LIN {X 0,Y 249.241,Z 277.058,A -85,B 0,C 180,E1 -19068.615,E2 -19068.615} C_VEL
LIN {X 0,Y 249.451,Z 277.034,A -85,B 0,C 180,E1 -19071.901,E2 -19071.901} C_VEL
LIN {X 0,Y 249.292,Z 277.04,A -85,B 0,C 180,E1 -19075.148,E2 -19075.148} C_VEL
LIN {X 0,Y 249.563,Z 277.018,A -85,B 0,C 180,E1 -19077.813,E2 -19077.813} C_VEL
LIN {X 0,Y 249.011,Z 277.095,A -85,B 0,C 180,E1 -19079.16,E2 -19079.16} C_VEL
LIN {X 0,Y 247.389,Z 277.302,A -85,B 0,C 180,E1 -19080.48,E2 -19080.48} C_VEL
LIN {X 0,Y 243.426,Z 277.789,A -85,B 0,C 180,E1 -19083.136,E2 -19083.136} C_VEL
LIN {X 0,Y 242.327,Z 277.917,A -85,B 0,C 180,E1 -19084.528,E2 -19084.528} C_VEL
LIN {X 0,Y 242.256,Z 277.921,A -85,B 0,C 180,E1 -19085,E2 -19085} C_VEL
LIN {X 0,Y 242.423,Z 277.913,A -85,B 0,C 180,E1 -19088.334,E2 -19088.334} C_VEL
LIN {X 0,Y 242.16,Z 277.946,A -85,B 0,C 180,E1 -19093.425,E2 -19093.425} C_VEL
LIN {X 0,Y 242.146,Z 277.937,A -85,B 0,C 180,E1 -19096.872,E2 -19096.872} C_VEL
LIN {X 0,Y 242.049,Z 277.953,A -85,B 0,C 180,E1 -19101.703,E2 -19101.703} C_VEL
LIN {X 0,Y 242.063,Z 277.952,A -85,B 0,C 180,E1 -19105.838,E2 -19105.838} C_VEL
LIN {X 0,Y 242.003,Z 277.929,A -85,B 0,C 180,E1 -19109.583,E2 -19109.583} C_VEL
LIN {X 0,Y 241.984,Z 277.969,A -85,B 0,C 180,E1 -19113.492,E2 -19113.492} C_VEL
LIN {X 0,Y 241.987,Z 277.941,A -85,B 0,C 180,E1 -19117.582,E2 -19117.582} C_VEL
LIN {X 0,Y 241.966,Z 278.133,A -85,B 0,C 180,E1 -19122.089,E2 -19122.089} C_VEL
LIN {X 0,Y 244.588,Z 286.288,A -85,B 0,C 180,E1 -19125.918,E2 -19125.918} C_VEL
LIN {X 0,Y 246.843,Z 293.756,A -85,B 0,C 180,E1 -19129.093,E2 -19129.093} C_VEL
LIN {X 0,Y 249.068,Z 301.648,A -85,B 0,C 180,E1 -19132.141,E2 -19132.141} C_VEL
LIN {X 0,Y 255.279,Z 314.084,A -85,B 0,C 180,E1 -19133.592,E2 -19133.592} C_VEL
LIN {X 0,Y 262.138,Z 329.274,A -85,B 0,C 180,E1 -19135.107,E2 -19135.107} C_VEL
LIN {X 0,Y 263.614,Z 333.202,A -85,B 0,C 180,E1 -19135.441,E2 -19135.441} C_VEL
LIN {X 0,Y 264.453,Z 341.441,A -85,B 0,C 180,E1 -19135.825,E2 -19135.825} C_VEL
LIN {X 0,Y 260.682,Z 430.839,A -85,B 0,C 180,E1 -19138.284,E2 -19138.284} C_VEL
LIN {X 0,Y 259.42,Z 445.087,A -85,B 0,C 180,E1 -19138.965,E2 -19138.965} C_VEL
LIN {X 0,Y 257.726,Z 458.762,A -85,B 0,C 180,E1 -19139.93,E2 -19139.93} C_VEL
LIN {X 0,Y 255.853,Z 470.591,A -85,B 0,C 180,E1 -19141.045,E2 -19141.045} C_VEL
LIN {X 0,Y 253.532,Z 483.66,A -85,B 0,C 180,E1 -19142.644,E2 -19142.644} C_VEL
LIN {X 0,Y 251.02,Z 495.578,A -85,B 0,C 180,E1 -19144.504,E2 -19144.504} C_VEL
LIN {X 0,Y 248.301,Z 506.631,A -85,B 0,C 180,E1 -19146.656,E2 -19146.656} C_VEL
LIN {X 0,Y 245.98,Z 516.527,A -85,B 0,C 180,E1 -19149.076,E2 -19149.076} C_VEL
LIN {X 0,Y 244.075,Z 524.668,A -85,B 0,C 180,E1 -19151.535,E2 -19151.535} C_VEL
LIN {X 0,Y 242.606,Z 531.385,A -85,B 0,C 180,E1 -19154.026,E2 -19154.026} C_VEL
LIN {X 0,Y 241.38,Z 536.896,A -85,B 0,C 180,E1 -19156.531,E2 -19156.531} C_VEL
LIN {X 0,Y 240.535,Z 541.36,A -85,B 0,C 180,E1 -19159.052,E2 -19159.052} C_VEL
LIN {X 0,Y 240.083,Z 544.873,A -85,B 0,C 180,E1 -19161.584,E2 -19161.584} C_VEL
LIN {X 0,Y 239.765,Z 548.121,A -85,B 0,C 180,E1 -19164.955,E2 -19164.955} C_VEL
LIN {X 0,Y 239.831,Z 549.889,A -85,B 0,C 180,E1 -19168.321,E2 -19168.321} C_VEL
LIN {X 0,Y 239.891,Z 550.231,A -85,B 0,C 180,E1 -19170,E2 -19170} C_VEL
LIN {X 0,Y 239.832,Z 550.21,A -85,B 0,C 180,E1 -19171.679,E2 -19171.679} C_VEL
LIN {X 0,Y 239.798,Z 549.093,A -85,B 0,C 180,E1 -19175.044,E2 -19175.044} C_VEL
LIN {X 0,Y 240.089,Z 546.53,A -85,B 0,C 180,E1 -19178.416,E2 -19178.416} C_VEL
LIN {X 0,Y 240.843,Z 542.397,A -85,B 0,C 180,E1 -19181.786,E2 -19181.786} C_VEL
LIN {X 0,Y 242.35,Z 536.619,A -85,B 0,C 180,E1 -19185.129,E2 -19185.129} C_VEL
LIN {X 0,Y 243.804,Z 531.335,A -85,B 0,C 180,E1 -19187.509,E2 -19187.509} C_VEL
LIN {X 0,Y 245.627,Z 524.336,A -85,B 0,C 180,E1 -19190.081,E2 -19190.081} C_VEL
LIN {X 0,Y 247.967,Z 516.181,A -85,B 0,C 180,E1 -19192.496,E2 -19192.496} C_VEL
LIN {X 0,Y 250.678,Z 506.282,A -85,B 0,C 180,E1 -19194.868,E2 -19194.868} C_VEL
LIN {X 0,Y 253.686,Z 495.218,A -85,B 0,C 180,E1 -19196.977,E2 -19196.977} C_VEL
LIN {X 0,Y 256.269,Z 483.685,A -85,B 0,C 180,E1 -19198.752,E2 -19198.752} C_VEL
LIN {X 0,Y 258.66,Z 471.958,A -85,B 0,C 180,E1 -19200.176,E2 -19200.176} C_VEL
LIN {X 0,Y 260.838,Z 459.44,A -85,B 0,C 180,E1 -19201.356,E2 -19201.356} C_VEL
LIN {X 0,Y 262.802,Z 445.333,A -85,B 0,C 180,E1 -19202.333,E2 -19202.333} C_VEL
LIN {X 0,Y 264.18,Z 431.307,A -85,B 0,C 180,E1 -19202.992,E2 -19202.992} C_VEL
LIN {X 0,Y 266.368,Z 384.252,A -85,B 0,C 180,E1 -19204.294,E2 -19204.294} C_VEL
LIN {X 0,Y 268.154,Z 341.465,A -85,B 0,C 180,E1 -19205.452,E2 -19205.452} C_VEL
LIN {X 0,Y 267.344,Z 337.375,A -85,B 0,C 180,E1 -19205.711,E2 -19205.711} C_VEL
LIN {X 0,Y 259.951,Z 321.227,A -85,B 0,C 180,E1 -19207.443,E2 -19207.443} C_VEL
LIN {X 0,Y 253.336,Z 308.74,A -85,B 0,C 180,E1 -19209.035,E2 -19209.035} C_VEL
LIN {X 0,Y 249.464,Z 301.565,A -85,B 0,C 180,E1 -19210.088,E2 -19210.088} C_VEL
LIN {X 0,Y 247.111,Z 293.383,A -85,B 0,C 180,E1 -19213.557,E2 -19213.557} C_VEL
LIN {X 0,Y 244.395,Z 285.114,A -85,B 0,C 180,E1 -19217.486,E2 -19217.486} C_VEL
LIN {X 0,Y 241.98,Z 278.041,A -85,B 0,C 180,E1 -19221.315,E2 -19221.315} C_VEL
LIN {X 0,Y 241.979,Z 277.937,A -85,B 0,C 180,E1 -19224.488,E2 -19224.488} C_VEL
LIN {X 0,Y 241.969,Z 277.942,A -85,B 0,C 180,E1 -19228.48,E2 -19228.48} C_VEL
LIN {X 0,Y 241.999,Z 277.945,A -85,B 0,C 180,E1 -19232.312,E2 -19232.312} C_VEL
LIN {X 0,Y 242.054,Z 277.949,A -85,B 0,C 180,E1 -19236.016,E2 -19236.016} C_VEL
LIN {X 0,Y 242.034,Z 277.949,A -85,B 0,C 180,E1 -19239.608,E2 -19239.608} C_VEL
LIN {X 0,Y 242.16,Z 277.933,A -85,B 0,C 180,E1 -19243.278,E2 -19243.278} C_VEL
LIN {X 0,Y 242.183,Z 277.928,A -85,B 0,C 180,E1 -19248.28,E2 -19248.28} C_VEL
LIN {X 0,Y 242.423,Z 277.902,A -85,B 0,C 180,E1 -19251.666,E2 -19251.666} C_VEL
LIN {X 0,Y 242.256,Z 277.934,A -85,B 0,C 180,E1 -19255.008,E2 -19255.008} C_VEL
LIN {X 0,Y 242.633,Z 277.875,A -85,B 0,C 180,E1 -19258.341,E2 -19258.341} C_VEL
LIN {X 0,Y 242.633,Z 277.873,A -85,B 0,C 180,E1 -19261.66,E2 -19261.66} C_VEL
LIN {X 0,Y 242.425,Z 277.898,A -85,B 0,C 180,E1 -19266.74,E2 -19266.74} C_VEL
LIN {X 0,Y 242.312,Z 277.923,A -85,B 0,C 180,E1 -19270.022,E2 -19270.022} C_VEL
LIN {X 0,Y 242.162,Z 277.935,A -85,B 0,C 180,E1 -19275.142,E2 -19275.142} C_VEL
LIN {X 0,Y 242.071,Z 277.953,A -85,B 0,C 180,E1 -19278.625,E2 -19278.625} C_VEL
LIN {X 0,Y 242.04,Z 277.961,A -85,B 0,C 180,E1 -19282.178,E2 -19282.178} C_VEL
LIN {X 0,Y 242.065,Z 277.959,A -85,B 0,C 180,E1 -19285.839,E2 -19285.839} C_VEL
LIN {X 0,Y 242.006,Z 277.929,A -85,B 0,C 180,E1 -19289.584,E2 -19289.584} C_VEL
LIN {X 0,Y 241.99,Z 277.948,A -85,B 0,C 180,E1 -19293.492,E2 -19293.492} C_VEL
LIN {X 0,Y 242.04,Z 278.135,A -85,B 0,C 180,E1 -19296.725,E2 -19296.725} C_VEL
LIN {X 0,Y 244.197,Z 284.736,A -85,B 0,C 180,E1 -19300.358,E2 -19300.358} C_VEL
LIN {X 0,Y 246.509,Z 292.185,A -85,B 0,C 180,E1 -19304.056,E2 -19304.056} C_VEL
LIN {X 0,Y 248.881,Z 300.613,A -85,B 0,C 180,E1 -19307.84,E2 -19307.84} C_VEL
LIN {X 0,Y 251.042,Z 309.201,A -85,B 0,C 180,E1 -19311.295,E2 -19311.295} C_VEL
LIN {X 0,Y 255.898,Z 318.813,A -85,B 0,C 180,E1 -19312.553,E2 -19312.553} C_VEL
LIN {X 0,Y 262.144,Z 332.18,A -85,B 0,C 180,E1 -19314.035,E2 -19314.035} C_VEL
LIN {X 0,Y 265.974,Z 354.542,A -85,B 0,C 180,E1 -19315.331,E2 -19315.331} C_VEL
LIN {X 0,Y 267.064,Z 362.449,A -85,B 0,C 180,E1 -19315.736,E2 -19315.736} C_VEL
LIN {X 0,Y 264.429,Z 427.598,A -85,B 0,C 180,E1 -19317.384,E2 -19317.384} C_VEL
LIN {X 0,Y 263.126,Z 441.134,A -85,B 0,C 180,E1 -19317.994,E2 -19317.994} C_VEL
LIN {X 0,Y 261.559,Z 453.539,A -85,B 0,C 180,E1 -19318.853,E2 -19318.853} C_VEL
LIN {X 0,Y 259.621,Z 465.602,A -85,B 0,C 180,E1 -19319.993,E2 -19319.993} C_VEL
LIN {X 0,Y 257.248,Z 477.352,A -85,B 0,C 180,E1 -19321.439,E2 -19321.439} C_VEL
LIN {X 0,Y 254.58,Z 488.124,A -85,B 0,C 180,E1 -19323.125,E2 -19323.125} C_VEL
LIN {X 0,Y 252.112,Z 496.99,A -85,B 0,C 180,E1 -19324.842,E2 -19324.842} C_VEL
LIN {X 0,Y 249.235,Z 506.656,A -85,B 0,C 180,E1 -19327.187,E2 -19327.187} C_VEL
LIN {X 0,Y 246.739,Z 514.484,A -85,B 0,C 180,E1 -19329.579,E2 -19329.579} C_VEL
LIN {X 0,Y 244.494,Z 521.732,A -85,B 0,C 180,E1 -19332.433,E2 -19332.433} C_VEL
LIN {X 0,Y 242.871,Z 526.644,A -85,B 0,C 180,E1 -19334.904,E2 -19334.904} C_VEL
LIN {X 0,Y 241.633,Z 530.504,A -85,B 0,C 180,E1 -19337.4,E2 -19337.4} C_VEL
LIN {X 0,Y 240.832,Z 533.375,A -85,B 0,C 180,E1 -19339.916,E2 -19339.916} C_VEL
LIN {X 0,Y 240.401,Z 534.808,A -85,B 0,C 180,E1 -19341.595,E2 -19341.595} C_VEL
LIN {X 0,Y 239.927,Z 536.499,A -85,B 0,C 180,E1 -19344.959,E2 -19344.959} C_VEL
LIN {X 0,Y 239.893,Z 536.763,A -85,B 0,C 180,E1 -19348.321,E2 -19348.321} C_VEL
LIN {X 0,Y 240.021,Z 535.601,A -85,B 0,C 180,E1 -19351.678,E2 -19351.678} C_VEL
LIN {X 0,Y 240.545,Z 532.914,A -85,B 0,C 180,E1 -19355.028,E2 -19355.028} C_VEL
LIN {X 0,Y 241.466,Z 528.685,A -85,B 0,C 180,E1 -19358.368,E2 -19358.368} C_VEL
LIN {X 0,Y 242.501,Z 524.336,A -85,B 0,C 180,E1 -19360.858,E2 -19360.858} C_VEL
LIN {X 0,Y 244.235,Z 517.869,A -85,B 0,C 180,E1 -19363.733,E2 -19363.733} C_VEL
LIN {X 0,Y 246.174,Z 510.872,A -85,B 0,C 180,E1 -19366.161,E2 -19366.161} C_VEL
LIN {X 0,Y 248.461,Z 502.247,A -85,B 0,C 180,E1 -19368.555,E2 -19368.555} C_VEL
LIN {X 0,Y 250.585,Z 493.496,A -85,B 0,C 180,E1 -19370.522,E2 -19370.522} C_VEL
LIN {X 0,Y 253.083,Z 482.799,A -85,B 0,C 180,E1 -19372.447,E2 -19372.447} C_VEL
LIN {X 0,Y 255.272,Z 472.208,A -85,B 0,C 180,E1 -19373.959,E2 -19373.959} C_VEL
LIN {X 0,Y 257.329,Z 460.555,A -85,B 0,C 180,E1 -19375.26,E2 -19375.26} C_VEL
LIN {X 0,Y 259.046,Z 447.27,A -85,B 0,C 180,E1 -19376.38,E2 -19376.38} C_VEL
LIN {X 0,Y 260.309,Z 434.324,A -85,B 0,C 180,E1 -19377.14,E2 -19377.14} C_VEL
LIN {X 0,Y 261.113,Z 420.968,A -85,B 0,C 180,E1 -19377.622,E2 -19377.622} C_VEL
LIN {X 0,Y 263.267,Z 359.223,A -85,B 0,C 180,E1 -19379.182,E2 -19379.182} C_VEL
LIN {X 0,Y 258.935,Z 330.912,A -85,B 0,C 180,E1 -19380.645,E2 -19380.645} C_VEL
LIN {X 0,Y 257.727,Z 325.251,A -85,B 0,C 180,E1 -19380.995,E2 -19380.995} C_VEL
LIN {X 0,Y 251.935,Z 312.605,A -85,B 0,C 180,E1 -19382.282,E2 -19382.282} C_VEL
LIN {X 0,Y 250.406,Z 309.097,A -85,B 0,C 180,E1 -19382.745,E2 -19382.745} C_VEL
LIN {X 0,Y 248.171,Z 299.259,A -85,B 0,C 180,E1 -19386.491,E2 -19386.491} C_VEL
LIN {X 0,Y 246.195,Z 291.901,A -85,B 0,C 180,E1 -19389.577,E2 -19389.577} C_VEL
LIN {X 0,Y 243.774,Z 283.733,A -85,B 0,C 180,E1 -19393.283,E2 -19393.283} C_VEL
LIN {X 0,Y 241.929,Z 278.066,A -85,B 0,C 180,E1 -19396.14,E2 -19396.14} C_VEL
LIN {X 0,Y 241.972,Z 277.94,A -85,B 0,C 180,E1 -19400.283,E2 -19400.283} C_VEL
LIN {X 0,Y 242.036,Z 277.938,A -85,B 0,C 180,E1 -19404.497,E2 -19404.497} C_VEL
LIN {X 0,Y 241.974,Z 277.952,A -85,B 0,C 180,E1 -19408.479,E2 -19408.479} C_VEL
LIN {X 0,Y 242.005,Z 277.955,A -85,B 0,C 180,E1 -19412.312,E2 -19412.312} C_VEL
LIN {X 0,Y 242.055,Z 277.946,A -85,B 0,C 180,E1 -19416.015,E2 -19416.015} C_VEL
LIN {X 0,Y 242.034,Z 277.95,A -85,B 0,C 180,E1 -19419.607,E2 -19419.607} C_VEL
LIN {X 0,Y 242.161,Z 277.943,A -85,B 0,C 180,E1 -19423.277,E2 -19423.277} C_VEL
LIN {X 0,Y 242.177,Z 277.941,A -85,B 0,C 180,E1 -19428.279,E2 -19428.279} C_VEL
LIN {X 0,Y 242.397,Z 277.911,A -85,B 0,C 180,E1 -19431.664,E2 -19431.664} C_VEL
LIN {X 0,Y 242.252,Z 277.917,A -85,B 0,C 180,E1 -19435.006,E2 -19435.006} C_VEL
LIN {X 0,Y 242.632,Z 277.887,A -85,B 0,C 180,E1 -19438.34,E2 -19438.34} C_VEL
LIN {X 0,Y 242.632,Z 277.874,A -85,B 0,C 180,E1 -19441.659,E2 -19441.659} C_VEL
LIN {X 0,Y 242.256,Z 277.921,A -85,B 0,C 180,E1 -19445,E2 -19445} C_VEL
LIN {X 0,Y 241.632,Z 277.997,A -85,B 0,C 180,E1 -19446.39,E2 -19446.39} C_VEL
LIN {X 0,Y 238.772,Z 278.367,A -85,B 0,C 180,E1 -19448.656,E2 -19448.656} C_VEL
LIN {X 0,Y 236.291,Z 278.67,A -85,B 0,C 180,E1 -19450.502,E2 -19450.502} C_VEL
LIN {X 0,Y 235.197,Z 278.801,A -85,B 0,C 180,E1 -19451.935,E2 -19451.935} C_VEL
LIN {X 0,Y 235.093,Z 278.814,A -85,B 0,C 180,E1 -19452.422,E2 -19452.422} C_VEL
LIN {X 0,Y 235.092,Z 278.816,A -85,B 0,C 180,E1 -19456.94,E2 -19456.94} C_VEL
LIN {X 0,Y 234.989,Z 278.835,A -85,B 0,C 180,E1 -19462.01,E2 -19462.01} C_VEL
LIN {X 0,Y 234.964,Z 278.843,A -85,B 0,C 180,E1 -19466.657,E2 -19466.657} C_VEL
LIN {X 0,Y 234.918,Z 278.807,A -85,B 0,C 180,E1 -19470.569,E2 -19470.569} C_VEL
LIN {X 0,Y 234.938,Z 278.837,A -85,B 0,C 180,E1 -19474.636,E2 -19474.636} C_VEL
LIN {X 0,Y 234.938,Z 278.836,A -85,B 0,C 180,E1 -19478.945,E2 -19478.945} C_VEL
LIN {X 0,Y 234.927,Z 279,A -85,B 0,C 180,E1 -19480.591,E2 -19480.591} C_VEL
LIN {X 0,Y 237.675,Z 287.447,A -85,B 0,C 180,E1 -19484.793,E2 -19484.793} C_VEL
LIN {X 0,Y 240.055,Z 295.257,A -85,B 0,C 180,E1 -19488.291,E2 -19488.291} C_VEL
LIN {X 0,Y 241.831,Z 301.626,A -85,B 0,C 180,E1 -19490.881,E2 -19490.881} C_VEL
LIN {X 0,Y 247.567,Z 312.725,A -85,B 0,C 180,E1 -19492.326,E2 -19492.326} C_VEL
LIN {X 0,Y 254.203,Z 326.888,A -85,B 0,C 180,E1 -19493.87,E2 -19493.87} C_VEL
LIN {X 0,Y 257.787,Z 335.652,A -85,B 0,C 180,E1 -19494.701,E2 -19494.701} C_VEL
LIN {X 0,Y 258.422,Z 342.678,A -85,B 0,C 180,E1 -19495.029,E2 -19495.029} C_VEL
LIN {X 0,Y 254.549,Z 430.59,A -85,B 0,C 180,E1 -19497.485,E2 -19497.485} C_VEL
LIN {X 0,Y 253.26,Z 444.905,A -85,B 0,C 180,E1 -19498.181,E2 -19498.181} C_VEL
LIN {X 0,Y 251.586,Z 458.043,A -85,B 0,C 180,E1 -19499.117,E2 -19499.117} C_VEL
LIN {X 0,Y 249.633,Z 470.006,A -85,B 0,C 180,E1 -19500.252,E2 -19500.252} C_VEL
LIN {X 0,Y 247.517,Z 481.582,A -85,B 0,C 180,E1 -19501.668,E2 -19501.668} C_VEL
LIN {X 0,Y 245.128,Z 492.852,A -85,B 0,C 180,E1 -19503.386,E2 -19503.386} C_VEL
LIN {X 0,Y 242.729,Z 502.481,A -85,B 0,C 180,E1 -19505.176,E2 -19505.176} C_VEL
LIN {X 0,Y 240.071,Z 513.133,A -85,B 0,C 180,E1 -19507.631,E2 -19507.631} C_VEL
LIN {X 0,Y 237.898,Z 521.847,A -85,B 0,C 180,E1 -19510.14,E2 -19510.14} C_VEL
LIN {X 0,Y 236.051,Z 530.078,A -85,B 0,C 180,E1 -19513.125,E2 -19513.125} C_VEL
LIN {X 0,Y 234.448,Z 536.636,A -85,B 0,C 180,E1 -19516.125,E2 -19516.125} C_VEL
LIN {X 0,Y 233.513,Z 541.115,A -85,B 0,C 180,E1 -19518.719,E2 -19518.719} C_VEL
LIN {X 0,Y 233.032,Z 544.637,A -85,B 0,C 180,E1 -19521.327,E2 -19521.327} C_VEL
LIN {X 0,Y 232.686,Z 547.903,A -85,B 0,C 180,E1 -19524.801,E2 -19524.801} C_VEL
LIN {X 0,Y 232.742,Z 549.683,A -85,B 0,C 180,E1 -19528.27,E2 -19528.27} C_VEL
LIN {X 0,Y 232.801,Z 550.03,A -85,B 0,C 180,E1 -19530,E2 -19530} C_VEL
LIN {X 0,Y 232.743,Z 550.014,A -85,B 0,C 180,E1 -19531.73,E2 -19531.73} C_VEL
LIN {X 0,Y 232.727,Z 548.907,A -85,B 0,C 180,E1 -19535.198,E2 -19535.198} C_VEL
LIN {X 0,Y 233.04,Z 546.354,A -85,B 0,C 180,E1 -19538.673,E2 -19538.673} C_VEL
LIN {X 0,Y 233.603,Z 543.401,A -85,B 0,C 180,E1 -19541.277,E2 -19541.277} C_VEL
LIN {X 0,Y 234.994,Z 538.1,A -85,B 0,C 180,E1 -19544.727,E2 -19544.727} C_VEL
LIN {X 0,Y 236.798,Z 531.843,A -85,B 0,C 180,E1 -19547.758,E2 -19547.758} C_VEL
LIN {X 0,Y 238.911,Z 524.193,A -85,B 0,C 180,E1 -19550.671,E2 -19550.671} C_VEL
LIN {X 0,Y 241.367,Z 516.044,A -85,B 0,C 180,E1 -19553.146,E2 -19553.146} C_VEL
LIN {X 0,Y 244.241,Z 506.152,A -85,B 0,C 180,E1 -19555.57,E2 -19555.57} C_VEL
LIN {X 0,Y 247.364,Z 495.091,A -85,B 0,C 180,E1 -19557.725,E2 -19557.725} C_VEL
LIN {X 0,Y 249.938,Z 484.008,A -85,B 0,C 180,E1 -19559.477,E2 -19559.477} C_VEL
LIN {X 0,Y 252.55,Z 471.826,A -85,B 0,C 180,E1 -19560.985,E2 -19560.985} C_VEL
LIN {X 0,Y 254.787,Z 459.295,A -85,B 0,C 180,E1 -19562.188,E2 -19562.188} C_VEL
LIN {X 0,Y 256.833,Z 445.162,A -85,B 0,C 180,E1 -19563.18,E2 -19563.18} C_VEL
LIN {X 0,Y 258.231,Z 431.077,A -85,B 0,C 180,E1 -19563.853,E2 -19563.853} C_VEL
LIN {X 0,Y 260.282,Z 389.795,A -85,B 0,C 180,E1 -19565.009,E2 -19565.009} C_VEL
LIN {X 0,Y 262.345,Z 342.506,A -85,B 0,C 180,E1 -19566.312,E2 -19566.312} C_VEL
LIN {X 0,Y 261.526,Z 339.663,A -85,B 0,C 180,E1 -19566.54,E2 -19566.54} C_VEL
LIN {X 0,Y 254.828,Z 324.845,A -85,B 0,C 180,E1 -19568.186,E2 -19568.186} C_VEL
LIN {X 0,Y 248.582,Z 312.995,A -85,B 0,C 180,E1 -19569.755,E2 -19569.755} C_VEL
LIN {X 0,Y 242.373,Z 301.792,A -85,B 0,C 180,E1 -19571.473,E2 -19571.473} C_VEL
LIN {X 0,Y 239.793,Z 293.359,A -85,B 0,C 180,E1 -19575.3,E2 -19575.3} C_VEL
LIN {X 0,Y 237.206,Z 285.476,A -85,B 0,C 180,E1 -19579.321,E2 -19579.321} C_VEL
LIN {X 0,Y 234.941,Z 278.936,A -85,B 0,C 180,E1 -19583.12,E2 -19583.12} C_VEL
LIN {X 0,Y 234.952,Z 278.836,A -85,B 0,C 180,E1 -19587.424,E2 -19587.424} C_VEL
LIN {X 0,Y 234.933,Z 278.811,A -85,B 0,C 180,E1 -19591.404,E2 -19591.404} C_VEL
LIN {X 0,Y 234.983,Z 278.829,A -85,B 0,C 180,E1 -19595.247,E2 -19595.247} C_VEL
LIN {X 0,Y 235.008,Z 278.826,A -85,B 0,C 180,E1 -19598.97,E2 -19598.97} C_VEL
LIN {X 0,Y 235.093,Z 278.814,A -85,B 0,C 180,E1 -19603.06,E2 -19603.06} C_VEL
LIN {X 0,Y 235.115,Z 278.808,A -85,B 0,C 180,E1 -19607.923,E2 -19607.923} C_VEL
LIN {X 0,Y 235.372,Z 278.783,A -85,B 0,C 180,E1 -19611.414,E2 -19611.414} C_VEL
LIN {X 0,Y 235.399,Z 278.772,A -85,B 0,C 180,E1 -19613.142,E2 -19613.142} C_VEL
LIN {X 0,Y 235.592,Z 278.751,A -85,B 0,C 180,E1 -19618.291,E2 -19618.291} C_VEL
LIN {X 0,Y 235.593,Z 278.749,A -85,B 0,C 180,E1 -19621.71,E2 -19621.71} C_VEL
LIN {X 0,Y 235.401,Z 278.773,A -85,B 0,C 180,E1 -19626.859,E2 -19626.859} C_VEL
LIN {X 0,Y 235.235,Z 278.8,A -85,B 0,C 180,E1 -19630.327,E2 -19630.327} C_VEL
LIN {X 0,Y 235.11,Z 278.811,A -85,B 0,C 180,E1 -19635.607,E2 -19635.607} C_VEL
LIN {X 0,Y 235.007,Z 278.827,A -85,B 0,C 180,E1 -19639.206,E2 -19639.206} C_VEL
LIN {X 0,Y 234.974,Z 278.835,A -85,B 0,C 180,E1 -19642.882,E2 -19642.882} C_VEL
LIN {X 0,Y 234.966,Z 278.829,A -85,B 0,C 180,E1 -19646.659,E2 -19646.659} C_VEL
LIN {X 0,Y 234.922,Z 278.819,A -85,B 0,C 180,E1 -19650.57,E2 -19650.57} C_VEL
LIN {X 0,Y 234.994,Z 278.983,A -85,B 0,C 180,E1 -19654.883,E2 -19654.883} C_VEL
LIN {X 0,Y 236.993,Z 285.114,A -85,B 0,C 180,E1 -19658.518,E2 -19658.518} C_VEL
LIN {X 0,Y 239.386,Z 292.518,A -85,B 0,C 180,E1 -19662.474,E2 -19662.474} C_VEL
LIN {X 0,Y 241.579,Z 300.156,A -85,B 0,C 180,E1 -19666.12,E2 -19666.12} C_VEL
LIN {X 0,Y 243.828,Z 308.833,A -85,B 0,C 180,E1 -19669.854,E2 -19669.854} C_VEL
LIN {X 0,Y 246.07,Z 313.241,A -85,B 0,C 180,E1 -19670.55,E2 -19670.55} C_VEL
LIN {X 0,Y 251.385,Z 323.656,A -85,B 0,C 180,E1 -19671.923,E2 -19671.923} C_VEL
LIN {X 0,Y 256.825,Z 335.628,A -85,B 0,C 180,E1 -19673.274,E2 -19673.274} C_VEL
LIN {X 0,Y 260.897,Z 360.658,A -85,B 0,C 180,E1 -19674.742,E2 -19674.742} C_VEL
LIN {X 0,Y 261.153,Z 363.958,A -85,B 0,C 180,E1 -19674.887,E2 -19674.887} C_VEL
LIN {X 0,Y 258.462,Z 427.939,A -85,B 0,C 180,E1 -19676.543,E2 -19676.543} C_VEL
LIN {X 0,Y 257.142,Z 441.238,A -85,B 0,C 180,E1 -19677.157,E2 -19677.157} C_VEL
LIN {X 0,Y 255.51,Z 453.635,A -85,B 0,C 180,E1 -19678.03,E2 -19678.03} C_VEL
LIN {X 0,Y 253.384,Z 466.279,A -85,B 0,C 180,E1 -19679.252,E2 -19679.252} C_VEL
LIN {X 0,Y 251.049,Z 477.45,A -85,B 0,C 180,E1 -19680.666,E2 -19680.666} C_VEL
LIN {X 0,Y 248.242,Z 488.229,A -85,B 0,C 180,E1 -19682.381,E2 -19682.381} C_VEL
LIN {X 0,Y 245.166,Z 498.866,A -85,B 0,C 180,E1 -19684.533,E2 -19684.533} C_VEL
LIN {X 0,Y 242.225,Z 508.225,A -85,B 0,C 180,E1 -19686.94,E2 -19686.94} C_VEL
LIN {X 0,Y 239.672,Z 515.759,A -85,B 0,C 180,E1 -19689.398,E2 -19689.398} C_VEL
LIN {X 0,Y 237.682,Z 521.875,A -85,B 0,C 180,E1 -19691.912,E2 -19691.912} C_VEL
LIN {X 0,Y 236.015,Z 526.796,A -85,B 0,C 180,E1 -19694.455,E2 -19694.455} C_VEL
LIN {X 0,Y 234.684,Z 530.665,A -85,B 0,C 180,E1 -19697.021,E2 -19697.021} C_VEL
LIN {X 0,Y 233.806,Z 533.545,A -85,B 0,C 180,E1 -19699.61,E2 -19699.61} C_VEL
LIN {X 0,Y 233.361,Z 534.986,A -85,B 0,C 180,E1 -19701.339,E2 -19701.339} C_VEL
LIN {X 0,Y 232.849,Z 536.689,A -85,B 0,C 180,E1 -19704.805,E2 -19704.805} C_VEL
LIN {X 0,Y 232.806,Z 536.964,A -85,B 0,C 180,E1 -19708.27,E2 -19708.27} C_VEL
LIN {X 0,Y 232.935,Z 535.819,A -85,B 0,C 180,E1 -19711.729,E2 -19711.729} C_VEL
LIN {X 0,Y 233.488,Z 533.147,A -85,B 0,C 180,E1 -19715.181,E2 -19715.181} C_VEL
LIN {X 0,Y 234.458,Z 528.932,A -85,B 0,C 180,E1 -19718.62,E2 -19718.62} C_VEL
LIN {X 0,Y 235.529,Z 524.601,A -85,B 0,C 180,E1 -19721.183,E2 -19721.183} C_VEL
LIN {X 0,Y 237.345,Z 518.163,A -85,B 0,C 180,E1 -19724.14,E2 -19724.14} C_VEL
LIN {X 0,Y 239.371,Z 511.195,A -85,B 0,C 180,E1 -19726.634,E2 -19726.634} C_VEL
LIN {X 0,Y 241.749,Z 502.602,A -85,B 0,C 180,E1 -19729.09,E2 -19729.09} C_VEL
LIN {X 0,Y 243.985,Z 493.89,A -85,B 0,C 180,E1 -19731.104,E2 -19731.104} C_VEL
LIN {X 0,Y 246.573,Z 483.245,A -85,B 0,C 180,E1 -19733.073,E2 -19733.073} C_VEL
LIN {X 0,Y 248.835,Z 472.726,A -85,B 0,C 180,E1 -19734.619,E2 -19734.619} C_VEL
LIN {X 0,Y 250.955,Z 461.225,A -85,B 0,C 180,E1 -19735.949,E2 -19735.949} C_VEL
LIN {X 0,Y 252.669,Z 448.796,A -85,B 0,C 180,E1 -19737.044,E2 -19737.044} C_VEL
LIN {X 0,Y 254.016,Z 436.001,A -85,B 0,C 180,E1 -19737.842,E2 -19737.842} C_VEL
LIN {X 0,Y 254.918,Z 422.901,A -85,B 0,C 180,E1 -19738.357,E2 -19738.357} C_VEL
LIN {X 0,Y 257.196,Z 359.986,A -85,B 0,C 180,E1 -19739.993,E2 -19739.993} C_VEL
LIN {X 0,Y 253.075,Z 332.654,A -85,B 0,C 180,E1 -19741.455,E2 -19741.455} C_VEL
LIN {X 0,Y 252.068,Z 327.951,A -85,B 0,C 180,E1 -19741.759,E2 -19741.759} C_VEL
LIN {X 0,Y 246.262,Z 315.466,A -85,B 0,C 180,E1 -19743.103,E2 -19743.103} C_VEL
LIN {X 0,Y 243.307,Z 309.18,A -85,B 0,C 180,E1 -19743.885,E2 -19743.885} C_VEL
LIN {X 0,Y 241.436,Z 301.083,A -85,B 0,C 180,E1 -19747.055,E2 -19747.055} C_VEL
LIN {X 0,Y 239.476,Z 293.679,A -85,B 0,C 180,E1 -19750.266,E2 -19750.266} C_VEL
LIN {X 0,Y 236.754,Z 284.661,A -85,B 0,C 180,E1 -19754.565,E2 -19754.565} C_VEL
LIN {X 0,Y 234.904,Z 278.908,A -85,B 0,C 180,E1 -19757.675,E2 -19757.675} C_VEL
LIN {X 0,Y 234.955,Z 278.817,A -85,B 0,C 180,E1 -19761.085,E2 -19761.085} C_VEL
LIN {X 0,Y 234.96,Z 278.808,A -85,B 0,C 180,E1 -19765.366,E2 -19765.366} C_VEL
LIN {X 0,Y 234.967,Z 278.842,A -85,B 0,C 180,E1 -19770.157,E2 -19770.157} C_VEL
LIN {X 0,Y 234.992,Z 278.839,A -85,B 0,C 180,E1 -19773.793,E2 -19773.793} C_VEL
LIN {X 0,Y 235.009,Z 278.831,A -85,B 0,C 180,E1 -19778.969,E2 -19778.969} C_VEL
LIN {X 0,Y 235.094,Z 278.825,A -85,B 0,C 180,E1 -19783.059,E2 -19783.059} C_VEL
LIN {X 0,Y 235.11,Z 278.824,A -85,B 0,C 180,E1 -19787.921,E2 -19787.921} C_VEL
LIN {X 0,Y 235.328,Z 278.787,A -85,B 0,C 180,E1 -19791.412,E2 -19791.412} C_VEL
LIN {X 0,Y 235.389,Z 278.788,A -85,B 0,C 180,E1 -19793.14,E2 -19793.14} C_VEL
LIN {X 0,Y 235.591,Z 278.765,A -85,B 0,C 180,E1 -19798.29,E2 -19798.29} C_VEL
LIN {X 0,Y 235.592,Z 278.751,A -85,B 0,C 180,E1 -19801.709,E2 -19801.709} C_VEL
LIN {X 0,Y 235.4,Z 278.774,A -85,B 0,C 180,E1 -19806.858,E2 -19806.858} C_VEL
LIN {X 0,Y 235.234,Z 278.794,A -85,B 0,C 180,E1 -19810.326,E2 -19810.326} C_VEL
LIN {X 0,Y 235.093,Z 278.814,A -85,B 0,C 180,E1 -19812.422,E2 -19812.422} C_VEL
LIN {X 0,Y 234.387,Z 278.915,A -85,B 0,C 180,E1 -19813.852,E2 -19813.852} C_VEL
LIN {X 0,Y 231.517,Z 279.268,A -85,B 0,C 180,E1 -19816.186,E2 -19816.186} C_VEL
LIN {X 0,Y 229.087,Z 279.574,A -85,B 0,C 180,E1 -19818.089,E2 -19818.089} C_VEL
LIN {X 0,Y 228.025,Z 279.698,A -85,B 0,C 180,E1 -19819.565,E2 -19819.565} C_VEL
LIN {X 0,Y 227.927,Z 279.707,A -85,B 0,C 180,E1 -19820.066,E2 -19820.066} C_VEL
LIN {X 0,Y 227.91,Z 279.715,A -85,B 0,C 180,E1 -19823.633,E2 -19823.633} C_VEL
LIN {X 0,Y 227.876,Z 279.719,A -85,B 0,C 180,E1 -19827.556,E2 -19827.556} C_VEL
LIN {X 0,Y 227.864,Z 279.692,A -85,B 0,C 180,E1 -19831.623,E2 -19831.623} C_VEL
LIN {X 0,Y 227.879,Z 279.698,A -85,B 0,C 180,E1 -19835.871,E2 -19835.871} C_VEL
LIN {X 0,Y 227.928,Z 279.96,A -85,B 0,C 180,E1 -19839.016,E2 -19839.016} C_VEL
LIN {X 0,Y 230.916,Z 289.1,A -85,B 0,C 180,E1 -19843.819,E2 -19843.819} C_VEL
LIN {X 0,Y 233.177,Z 296.389,A -85,B 0,C 180,E1 -19847.268,E2 -19847.268} C_VEL
LIN {X 0,Y 234.73,Z 301.974,A -85,B 0,C 180,E1 -19849.607,E2 -19849.607} C_VEL
LIN {X 0,Y 241.502,Z 314.663,A -85,B 0,C 180,E1 -19851.369,E2 -19851.369} C_VEL
LIN {X 0,Y 248.702,Z 329.96,A -85,B 0,C 180,E1 -19853.124,E2 -19853.124} C_VEL
LIN {X 0,Y 251.971,Z 337.774,A -85,B 0,C 180,E1 -19853.909,E2 -19853.909} C_VEL
LIN {X 0,Y 252.44,Z 343.76,A -85,B 0,C 180,E1 -19854.188,E2 -19854.188} C_VEL
LIN {X 0,Y 248.47,Z 430.334,A -85,B 0,C 180,E1 -19856.648,E2 -19856.648} C_VEL
LIN {X 0,Y 247.249,Z 443.966,A -85,B 0,C 180,E1 -19857.312,E2 -19857.312} C_VEL
LIN {X 0,Y 245.662,Z 456.191,A -85,B 0,C 180,E1 -19858.166,E2 -19858.166} C_VEL
LIN {X 0,Y 243.469,Z 469.423,A -85,B 0,C 180,E1 -19859.419,E2 -19859.419} C_VEL
LIN {X 0,Y 241.043,Z 482.136,A -85,B 0,C 180,E1 -19861.009,E2 -19861.009} C_VEL
LIN {X 0,Y 238.485,Z 493.609,A -85,B 0,C 180,E1 -19862.821,E2 -19862.821} C_VEL
LIN {X 0,Y 235.737,Z 504.074,A -85,B 0,C 180,E1 -19864.86,E2 -19864.86} C_VEL
LIN {X 0,Y 233.057,Z 514.358,A -85,B 0,C 180,E1 -19867.389,E2 -19867.389} C_VEL
LIN {X 0,Y 230.827,Z 522.808,A -85,B 0,C 180,E1 -19869.969,E2 -19869.969} C_VEL
LIN {X 0,Y 228.926,Z 530.828,A -85,B 0,C 180,E1 -19873.044,E2 -19873.044} C_VEL
LIN {X 0,Y 227.5,Z 536.375,A -85,B 0,C 180,E1 -19875.692,E2 -19875.692} C_VEL
LIN {X 0,Y 226.509,Z 540.87,A -85,B 0,C 180,E1 -19878.365,E2 -19878.365} C_VEL
LIN {X 0,Y 225.975,Z 544.4,A -85,B 0,C 180,E1 -19881.054,E2 -19881.054} C_VEL
LIN {X 0,Y 225.733,Z 546.241,A -85,B 0,C 180,E1 -19882.846,E2 -19882.846} C_VEL
LIN {X 0,Y 225.55,Z 548.76,A -85,B 0,C 180,E1 -19886.427,E2 -19886.427} C_VEL
LIN {X 0,Y 225.636,Z 549.476,A -85,B 0,C 180,E1 -19888.215,E2 -19888.215} C_VEL
LIN {X 0,Y 225.714,Z 549.829,A -85,B 0,C 180,E1 -19890,E2 -19890} C_VEL
LIN {X 0,Y 225.637,Z 549.817,A -85,B 0,C 180,E1 -19891.785,E2 -19891.785} C_VEL
LIN {X 0,Y 225.64,Z 548.72,A -85,B 0,C 180,E1 -19895.362,E2 -19895.362} C_VEL
LIN {X 0,Y 225.986,Z 546.178,A -85,B 0,C 180,E1 -19898.946,E2 -19898.946} C_VEL
LIN {X 0,Y 226.594,Z 543.232,A -85,B 0,C 180,E1 -19901.631,E2 -19901.631} C_VEL
LIN {X 0,Y 228.084,Z 537.941,A -85,B 0,C 180,E1 -19905.183,E2 -19905.183} C_VEL
LIN {X 0,Y 230.115,Z 531.066,A -85,B 0,C 180,E1 -19908.573,E2 -19908.573} C_VEL
LIN {X 0,Y 232.628,Z 522.802,A -85,B 0,C 180,E1 -19911.721,E2 -19911.721} C_VEL
LIN {X 0,Y 235.297,Z 514.405,A -85,B 0,C 180,E1 -19914.248,E2 -19914.248} C_VEL
LIN {X 0,Y 238.43,Z 504.207,A -85,B 0,C 180,E1 -19916.712,E2 -19916.712} C_VEL
LIN {X 0,Y 241.373,Z 493.828,A -85,B 0,C 180,E1 -19918.713,E2 -19918.713} C_VEL
LIN {X 0,Y 244.007,Z 482.89,A -85,B 0,C 180,E1 -19920.435,E2 -19920.435} C_VEL
LIN {X 0,Y 246.809,Z 469.926,A -85,B 0,C 180,E1 -19922.029,E2 -19922.029} C_VEL
LIN {X 0,Y 249.188,Z 456.901,A -85,B 0,C 180,E1 -19923.244,E2 -19923.244} C_VEL
LIN {X 0,Y 251.238,Z 442.717,A -85,B 0,C 180,E1 -19924.2,E2 -19924.2} C_VEL
LIN {X 0,Y 252.485,Z 429.653,A -85,B 0,C 180,E1 -19924.793,E2 -19924.793} C_VEL
LIN {X 0,Y 256.557,Z 345.746,A -85,B 0,C 180,E1 -19927.138,E2 -19927.138} C_VEL
LIN {X 0,Y 256.471,Z 343.541,A -85,B 0,C 180,E1 -19927.231,E2 -19927.231} C_VEL
LIN {X 0,Y 249.83,Z 328.641,A -85,B 0,C 180,E1 -19928.939,E2 -19928.939} C_VEL
LIN {X 0,Y 242.408,Z 314.491,A -85,B 0,C 180,E1 -19930.902,E2 -19930.902} C_VEL
LIN {X 0,Y 237.027,Z 305.289,A -85,B 0,C 180,E1 -19932.398,E2 -19932.398} C_VEL
LIN {X 0,Y 235.191,Z 301.931,A -85,B 0,C 180,E1 -19933.019,E2 -19933.019} C_VEL
LIN {X 0,Y 233.036,Z 294.954,A -85,B 0,C 180,E1 -19936.368,E2 -19936.368} C_VEL
LIN {X 0,Y 230.635,Z 287.822,A -85,B 0,C 180,E1 -19940.215,E2 -19940.215} C_VEL
LIN {X 0,Y 228.273,Z 281.258,A -85,B 0,C 180,E1 -19944.2,E2 -19944.2} C_VEL
LIN {X 0,Y 227.893,Z 279.794,A -85,B 0,C 180,E1 -19945.214,E2 -19945.214} C_VEL
LIN {X 0,Y 227.901,Z 279.68,A -85,B 0,C 180,E1 -19950.436,E2 -19950.436} C_VEL
LIN {X 0,Y 227.925,Z 279.714,A -85,B 0,C 180,E1 -19954.426,E2 -19954.426} C_VEL
LIN {X 0,Y 227.959,Z 279.709,A -85,B 0,C 180,E1 -19958.287,E2 -19958.287} C_VEL
LIN {X 0,Y 228.031,Z 279.695,A -85,B 0,C 180,E1 -19962.826,E2 -19962.826} C_VEL
LIN {X 0,Y 228.072,Z 279.687,A -85,B 0,C 180,E1 -19967.544,E2 -19967.544} C_VEL
LIN {X 0,Y 228.302,Z 279.667,A -85,B 0,C 180,E1 -19971.146,E2 -19971.146} C_VEL
LIN {X 0,Y 228.35,Z 279.649,A -85,B 0,C 180,E1 -19972.929,E2 -19972.929} C_VEL
LIN {X 0,Y 228.551,Z 279.628,A -85,B 0,C 180,E1 -19978.238,E2 -19978.238} C_VEL
LIN {X 0,Y 228.551,Z 279.626,A -85,B 0,C 180,E1 -19981.763,E2 -19981.763} C_VEL
LIN {X 0,Y 228.352,Z 279.65,A -85,B 0,C 180,E1 -19987.072,E2 -19987.072} C_VEL
LIN {X 0,Y 228.157,Z 279.678,A -85,B 0,C 180,E1 -19990.651,E2 -19990.651} C_VEL
LIN {X 0,Y 228.061,Z 279.699,A -85,B 0,C 180,E1 -19994.273,E2 -19994.273} C_VEL
LIN {X 0,Y 228.001,Z 279.71,A -85,B 0,C 180,E1 -19997.954,E2 -19997.954} C_VEL
LIN {X 0,Y 227.952,Z 279.715,A -85,B 0,C 180,E1 -20002.344,E2 -20002.344} C_VEL
LIN {X 0,Y 227.941,Z 279.703,A -85,B 0,C 180,E1 -20006.603,E2 -20006.603} C_VEL
LIN {X 0,Y 227.896,Z 279.69,A -85,B 0,C 180,E1 -20010.292,E2 -20010.292} C_VEL
LIN {X 0,Y 227.96,Z 279.941,A -85,B 0,C 180,E1 -20012.915,E2 -20012.915} C_VEL
LIN {X 0,Y 230.022,Z 285.881,A -85,B 0,C 180,E1 -20016.751,E2 -20016.751} C_VEL
LIN {X 0,Y 232.284,Z 293.112,A -85,B 0,C 180,E1 -20020.853,E2 -20020.853} C_VEL
LIN {X 0,Y 234.59,Z 300.745,A -85,B 0,C 180,E1 -20024.751,E2 -20024.751} C_VEL
LIN {X 0,Y 236.735,Z 308.899,A -85,B 0,C 180,E1 -20028.425,E2 -20028.425} C_VEL
LIN {X 0,Y 244.381,Z 323.185,A -85,B 0,C 180,E1 -20030.59,E2 -20030.59} C_VEL
LIN {X 0,Y 251.338,Z 338.057,A -85,B 0,C 180,E1 -20032.407,E2 -20032.407} C_VEL
LIN {X 0,Y 255.13,Z 361.799,A -85,B 0,C 180,E1 -20033.85,E2 -20033.85} C_VEL
LIN {X 0,Y 255.351,Z 365.68,A -85,B 0,C 180,E1 -20034.013,E2 -20034.013} C_VEL
LIN {X 0,Y 252.618,Z 427.25,A -85,B 0,C 180,E1 -20035.621,E2 -20035.621} C_VEL
LIN {X 0,Y 251.333,Z 440.574,A -85,B 0,C 180,E1 -20036.237,E2 -20036.237} C_VEL
LIN {X 0,Y 249.51,Z 453.731,A -85,B 0,C 180,E1 -20037.166,E2 -20037.166} C_VEL
LIN {X 0,Y 247.499,Z 465.329,A -85,B 0,C 180,E1 -20038.296,E2 -20038.296} C_VEL
LIN {X 0,Y 245.221,Z 476.168,A -85,B 0,C 180,E1 -20039.66,E2 -20039.66} C_VEL
LIN {X 0,Y 242.319,Z 487.27,A -85,B 0,C 180,E1 -20041.41,E2 -20041.41} C_VEL
LIN {X 0,Y 239.303,Z 497.214,A -85,B 0,C 180,E1 -20043.393,E2 -20043.393} C_VEL
LIN {X 0,Y 236.212,Z 506.895,A -85,B 0,C 180,E1 -20045.852,E2 -20045.852} C_VEL
LIN {X 0,Y 233.415,Z 514.742,A -85,B 0,C 180,E1 -20048.356,E2 -20048.356} C_VEL
LIN {X 0,Y 231.575,Z 520.106,A -85,B 0,C 180,E1 -20050.498,E2 -20050.498} C_VEL
LIN {X 0,Y 229.722,Z 525.412,A -85,B 0,C 180,E1 -20053.104,E2 -20053.104} C_VEL
LIN {X 0,Y 228.098,Z 529.623,A -85,B 0,C 180,E1 -20055.73,E2 -20055.73} C_VEL
LIN {X 0,Y 226.801,Z 533.714,A -85,B 0,C 180,E1 -20059.285,E2 -20059.285} C_VEL
LIN {X 0,Y 226.32,Z 535.163,A -85,B 0,C 180,E1 -20061.068,E2 -20061.068} C_VEL
LIN {X 0,Y 225.773,Z 536.879,A -85,B 0,C 180,E1 -20064.642,E2 -20064.642} C_VEL
LIN {X 0,Y 225.72,Z 537.166,A -85,B 0,C 180,E1 -20068.216,E2 -20068.216} C_VEL
LIN {X 0,Y 225.852,Z 536.037,A -85,B 0,C 180,E1 -20071.783,E2 -20071.783} C_VEL
LIN {X 0,Y 226.435,Z 533.38,A -85,B 0,C 180,E1 -20075.343,E2 -20075.343} C_VEL
LIN {X 0,Y 227.441,Z 529.18,A -85,B 0,C 180,E1 -20078.888,E2 -20078.888} C_VEL
LIN {X 0,Y 228.579,Z 524.866,A -85,B 0,C 180,E1 -20081.528,E2 -20081.528} C_VEL
LIN {X 0,Y 230.483,Z 518.454,A -85,B 0,C 180,E1 -20084.57,E2 -20084.57} C_VEL
LIN {X 0,Y 232.592,Z 511.518,A -85,B 0,C 180,E1 -20087.134,E2 -20087.134} C_VEL
LIN {X 0,Y 235.069,Z 502.956,A -85,B 0,C 180,E1 -20089.654,E2 -20089.654} C_VEL
LIN {X 0,Y 237.409,Z 494.284,A -85,B 0,C 180,E1 -20091.717,E2 -20091.717} C_VEL
LIN {X 0,Y 240.08,Z 483.692,A -85,B 0,C 180,E1 -20093.735,E2 -20093.735} C_VEL
LIN {X 0,Y 242.434,Z 473.243,A -85,B 0,C 180,E1 -20095.314,E2 -20095.314} C_VEL
LIN {X 0,Y 244.608,Z 461.86,A -85,B 0,C 180,E1 -20096.675,E2 -20096.675} C_VEL
LIN {X 0,Y 246.339,Z 450.231,A -85,B 0,C 180,E1 -20097.746,E2 -20097.746} C_VEL
LIN {X 0,Y 247.799,Z 437.363,A -85,B 0,C 180,E1 -20098.594,E2 -20098.594} C_VEL
LIN {X 0,Y 248.814,Z 423.411,A -85,B 0,C 180,E1 -20099.174,E2 -20099.174} C_VEL
LIN {X 0,Y 251.208,Z 360.984,A -85,B 0,C 180,E1 -20100.83,E2 -20100.83} C_VEL
LIN {X 0,Y 246.894,Z 331.846,A -85,B 0,C 180,E1 -20102.446,E2 -20102.446} C_VEL
LIN {X 0,Y 241.623,Z 320.228,A -85,B 0,C 180,E1 -20103.725,E2 -20103.725} C_VEL
LIN {X 0,Y 236.19,Z 309.016,A -85,B 0,C 180,E1 -20105.169,E2 -20105.169} C_VEL
LIN {X 0,Y 234.164,Z 300.475,A -85,B 0,C 180,E1 -20108.707,E2 -20108.707} C_VEL
LIN {X 0,Y 231.961,Z 292.755,A -85,B 0,C 180,E1 -20112.304,E2 -20112.304} C_VEL
LIN {X 0,Y 230.085,Z 286.718,A -85,B 0,C 180,E1 -20115.368,E2 -20115.368} C_VEL
LIN {X 0,Y 227.865,Z 279.784,A -85,B 0,C 180,E1 -20119.31,E2 -20119.31} C_VEL
LIN {X 0,Y 227.899,Z 279.703,A -85,B 0,C 180,E1 -20124.131,E2 -20124.131} C_VEL
LIN {X 0,Y 227.871,Z 279.704,A -85,B 0,C 180,E1 -20128.377,E2 -20128.377} C_VEL
LIN {X 0,Y 227.884,Z 279.715,A -85,B 0,C 180,E1 -20132.444,E2 -20132.444} C_VEL
LIN {X 0,Y 227.912,Z 279.708,A -85,B 0,C 180,E1 -20136.366,E2 -20136.366} C_VEL
LIN {X 0,Y 227.94,Z 279.703,A -85,B 0,C 180,E1 -20140.174,E2 -20140.174} C_VEL
LIN {X 0,Y 228.054,Z 279.693,A -85,B 0,C 180,E1 -20143.897,E2 -20143.897} C_VEL
LIN {X 0,Y 228.068,Z 279.701,A -85,B 0,C 180,E1 -20147.542,E2 -20147.542} C_VEL
LIN {X 0,Y 228.264,Z 279.664,A -85,B 0,C 180,E1 -20151.144,E2 -20151.144} C_VEL
LIN {X 0,Y 228.336,Z 279.668,A -85,B 0,C 180,E1 -20152.927,E2 -20152.927} C_VEL
LIN {X 0,Y 228.55,Z 279.642,A -85,B 0,C 180,E1 -20158.237,E2 -20158.237} C_VEL
LIN {X 0,Y 228.551,Z 279.628,A -85,B 0,C 180,E1 -20161.762,E2 -20161.762} C_VEL
LIN {X 0,Y 228.351,Z 279.654,A -85,B 0,C 180,E1 -20167.071,E2 -20167.071} C_VEL
LIN {X 0,Y 228.155,Z 279.674,A -85,B 0,C 180,E1 -20170.65,E2 -20170.65} C_VEL
LIN {X 0,Y 228.059,Z 279.699,A -85,B 0,C 180,E1 -20174.272,E2 -20174.272} C_VEL
LIN {X 0,Y 227.999,Z 279.709,A -85,B 0,C 180,E1 -20177.953,E2 -20177.953} C_VEL
LIN {X 0,Y 227.927,Z 279.707,A -85,B 0,C 180,E1 -20180.066,E2 -20180.066} C_VEL
LIN {X 0,Y 227.23,Z 279.799,A -85,B 0,C 180,E1 -20181.54,E2 -20181.54} C_VEL
LIN {X 0,Y 224.378,Z 280.16,A -85,B 0,C 180,E1 -20183.946,E2 -20183.946} C_VEL
LIN {X 0,Y 221.965,Z 280.463,A -85,B 0,C 180,E1 -20185.908,E2 -20185.908} C_VEL
LIN {X 0,Y 220.919,Z 280.586,A -85,B 0,C 180,E1 -20187.432,E2 -20187.432} C_VEL
LIN {X 0,Y 220.827,Z 280.584,A -85,B 0,C 180,E1 -20187.948,E2 -20187.948} C_VEL
LIN {X 0,Y 220.835,Z 280.561,A -85,B 0,C 180,E1 -20190.768,E2 -20190.768} C_VEL
LIN {X 0,Y 220.8,Z 280.59,A -85,B 0,C 180,E1 -20194.955,E2 -20194.955} C_VEL
LIN {X 0,Y 220.848,Z 280.826,A -85,B 0,C 180,E1 -20197.202,E2 -20197.202} C_VEL
LIN {X 0,Y 223.283,Z 288.098,A -85,B 0,C 180,E1 -20201.375,E2 -20201.375} C_VEL
LIN {X 0,Y 225.953,Z 296.519,A -85,B 0,C 180,E1 -20205.674,E2 -20205.674} C_VEL
LIN {X 0,Y 227.608,Z 302.185,A -85,B 0,C 180,E1 -20208.197,E2 -20208.197} C_VEL
LIN {X 0,Y 234.644,Z 315.005,A -85,B 0,C 180,E1 -20210.141,E2 -20210.141} C_VEL
LIN {X 0,Y 242.198,Z 330.697,A -85,B 0,C 180,E1 -20212.081,E2 -20212.081} C_VEL
LIN {X 0,Y 246.27,Z 340.399,A -85,B 0,C 180,E1 -20213.109,E2 -20213.109} C_VEL
LIN {X 0,Y 246.511,Z 344.831,A -85,B 0,C 180,E1 -20213.307,E2 -20213.307} C_VEL
LIN {X 0,Y 242.448,Z 430.067,A -85,B 0,C 180,E1 -20215.769,E2 -20215.769} C_VEL
LIN {X 0,Y 241.198,Z 443.783,A -85,B 0,C 180,E1 -20216.448,E2 -20216.448} C_VEL
LIN {X 0,Y 239.459,Z 456.602,A -85,B 0,C 180,E1 -20217.365,E2 -20217.365} C_VEL
LIN {X 0,Y 237.355,Z 468.838,A -85,B 0,C 180,E1 -20218.543,E2 -20218.543} C_VEL
LIN {X 0,Y 234.785,Z 481.803,A -85,B 0,C 180,E1 -20220.187,E2 -20220.187} C_VEL
LIN {X 0,Y 232.133,Z 493.178,A -85,B 0,C 180,E1 -20222.014,E2 -20222.014} C_VEL
LIN {X 0,Y 229.304,Z 503.695,A -85,B 0,C 180,E1 -20224.104,E2 -20224.104} C_VEL
LIN {X 0,Y 226.91,Z 512.446,A -85,B 0,C 180,E1 -20226.257,E2 -20226.257} C_VEL
LIN {X 0,Y 224.459,Z 521.226,A -85,B 0,C 180,E1 -20228.896,E2 -20228.896} C_VEL
LIN {X 0,Y 222.568,Z 528.456,A -85,B 0,C 180,E1 -20231.593,E2 -20231.593} C_VEL
LIN {X 0,Y 221.033,Z 534.395,A -85,B 0,C 180,E1 -20234.32,E2 -20234.32} C_VEL
LIN {X 0,Y 219.774,Z 539.221,A -85,B 0,C 180,E1 -20237.065,E2 -20237.065} C_VEL
LIN {X 0,Y 218.937,Z 544.163,A -85,B 0,C 180,E1 -20240.764,E2 -20240.764} C_VEL
LIN {X 0,Y 218.499,Z 547.466,A -85,B 0,C 180,E1 -20244.463,E2 -20244.463} C_VEL
LIN {X 0,Y 218.532,Z 549.268,A -85,B 0,C 180,E1 -20248.157,E2 -20248.157} C_VEL
LIN {X 0,Y 218.629,Z 549.628,A -85,B 0,C 180,E1 -20250,E2 -20250} C_VEL
LIN {X 0,Y 218.497,Z 549.256,A -85,B 0,C 180,E1 -20253.688,E2 -20253.688} C_VEL
LIN {X 0,Y 218.561,Z 548.534,A -85,B 0,C 180,E1 -20255.536,E2 -20255.536} C_VEL
LIN {X 0,Y 218.949,Z 546.001,A -85,B 0,C 180,E1 -20259.236,E2 -20259.236} C_VEL
LIN {X 0,Y 219.875,Z 541.902,A -85,B 0,C 180,E1 -20262.929,E2 -20262.929} C_VEL
LIN {X 0,Y 221.189,Z 537.782,A -85,B 0,C 180,E1 -20265.669,E2 -20265.669} C_VEL
LIN {X 0,Y 222.864,Z 532.607,A -85,B 0,C 180,E1 -20268.382,E2 -20268.382} C_VEL
LIN {X 0,Y 225.189,Z 525.154,A -85,B 0,C 180,E1 -20271.513,E2 -20271.513} C_VEL
LIN {X 0,Y 227.814,Z 517.275,A -85,B 0,C 180,E1 -20274.127,E2 -20274.127} C_VEL
LIN {X 0,Y 230.89,Z 507.691,A -85,B 0,C 180,E1 -20276.677,E2 -20276.677} C_VEL
LIN {X 0,Y 233.887,Z 498.069,A -85,B 0,C 180,E1 -20278.736,E2 -20278.736} C_VEL
LIN {X 0,Y 236.901,Z 486.628,A -85,B 0,C 180,E1 -20280.73,E2 -20280.73} C_VEL
LIN {X 0,Y 239.739,Z 474.848,A -85,B 0,C 180,E1 -20282.344,E2 -20282.344} C_VEL
LIN {X 0,Y 242.493,Z 461.223,A -85,B 0,C 180,E1 -20283.786,E2 -20283.786} C_VEL
LIN {X 0,Y 244.669,Z 447.856,A -85,B 0,C 180,E1 -20284.812,E2 -20284.812} C_VEL
LIN {X 0,Y 246.321,Z 433.999,A -85,B 0,C 180,E1 -20285.544,E2 -20285.544} C_VEL
LIN {X 0,Y 247.471,Z 416.592,A -85,B 0,C 180,E1 -20286.106,E2 -20286.106} C_VEL
LIN {X 0,Y 250.808,Z 345.883,A -85,B 0,C 180,E1 -20288.12,E2 -20288.12} C_VEL
LIN {X 0,Y 244.15,Z 330.905,A -85,B 0,C 180,E1 -20289.92,E2 -20289.92} C_VEL
LIN {X 0,Y 236.701,Z 316.893,A -85,B 0,C 180,E1 -20291.993,E2 -20291.993} C_VEL
LIN {X 0,Y 230.735,Z 306.623,A -85,B 0,C 180,E1 -20293.762,E2 -20293.762} C_VEL
LIN {X 0,Y 228.108,Z 302.208,A -85,B 0,C 180,E1 -20294.642,E2 -20294.642} C_VEL
LIN {X 0,Y 225.365,Z 293.699,A -85,B 0,C 180,E1 -20299.09,E2 -20299.09} C_VEL
LIN {X 0,Y 223.006,Z 286.805,A -85,B 0,C 180,E1 -20303.218,E2 -20303.218} C_VEL
LIN {X 0,Y 221.815,Z 283.416,A -85,B 0,C 180,E1 -20305.464,E2 -20305.464} C_VEL
LIN {X 0,Y 220.813,Z 280.681,A -85,B 0,C 180,E1 -20307.515,E2 -20307.515} C_VEL
LIN {X 0,Y 220.824,Z 280.567,A -85,B 0,C 180,E1 -20311.485,E2 -20311.485} C_VEL
LIN {X 0,Y 220.864,Z 280.587,A -85,B 0,C 180,E1 -20315.565,E2 -20315.565} C_VEL
LIN {X 0,Y 220.889,Z 280.582,A -85,B 0,C 180,E1 -20319.514,E2 -20319.514} C_VEL
LIN {X 0,Y 221.013,Z 280.566,A -85,B 0,C 180,E1 -20323.371,E2 -20323.371} C_VEL
LIN {X 0,Y 221.104,Z 280.555,A -85,B 0,C 180,E1 -20329.006,E2 -20329.006} C_VEL
LIN {X 0,Y 221.285,Z 280.529,A -85,B 0,C 180,E1 -20332.702,E2 -20332.702} C_VEL
LIN {X 0,Y 221.509,Z 280.504,A -85,B 0,C 180,E1 -20338.182,E2 -20338.182} C_VEL
LIN {X 0,Y 221.51,Z 280.502,A -85,B 0,C 180,E1 -20341.819,E2 -20341.819} C_VEL
LIN {X 0,Y 221.287,Z 280.53,A -85,B 0,C 180,E1 -20347.299,E2 -20347.299} C_VEL
LIN {X 0,Y 221.104,Z 280.554,A -85,B 0,C 180,E1 -20350.995,E2 -20350.995} C_VEL
LIN {X 0,Y 221.014,Z 280.568,A -85,B 0,C 180,E1 -20356.631,E2 -20356.631} C_VEL
LIN {X 0,Y 220.898,Z 280.583,A -85,B 0,C 180,E1 -20360.486,E2 -20360.486} C_VEL
LIN {X 0,Y 220.87,Z 280.589,A -85,B 0,C 180,E1 -20364.435,E2 -20364.435} C_VEL
LIN {X 0,Y 220.826,Z 280.564,A -85,B 0,C 180,E1 -20368.516,E2 -20368.516} C_VEL
LIN {X 0,Y 220.868,Z 280.803,A -85,B 0,C 180,E1 -20370.606,E2 -20370.606} C_VEL
LIN {X 0,Y 222.905,Z 286.347,A -85,B 0,C 180,E1 -20374.579,E2 -20374.579} C_VEL
LIN {X 0,Y 224.593,Z 291.623,A -85,B 0,C 180,E1 -20377.869,E2 -20377.869} C_VEL
LIN {X 0,Y 226.831,Z 298.878,A -85,B 0,C 180,E1 -20381.962,E2 -20381.962} C_VEL
LIN {X 0,Y 228.814,Z 306,A -85,B 0,C 180,E1 -20385.572,E2 -20385.572} C_VEL
LIN {X 0,Y 229.681,Z 308.972,A -85,B 0,C 180,E1 -20386.853,E2 -20386.853} C_VEL
LIN {X 0,Y 237.584,Z 323.326,A -85,B 0,C 180,E1 -20389.218,E2 -20389.218} C_VEL
LIN {X 0,Y 243.151,Z 334.696,A -85,B 0,C 180,E1 -20390.77,E2 -20390.77} C_VEL
LIN {X 0,Y 246.123,Z 341.578,A -85,B 0,C 180,E1 -20391.581,E2 -20391.581} C_VEL
LIN {X 0,Y 249.675,Z 364.685,A -85,B 0,C 180,E1 -20393.019,E2 -20393.019} C_VEL
LIN {X 0,Y 246.798,Z 427.62,A -85,B 0,C 180,E1 -20394.703,E2 -20394.703} C_VEL
LIN {X 0,Y 245.371,Z 441.451,A -85,B 0,C 180,E1 -20395.364,E2 -20395.364} C_VEL
LIN {X 0,Y 243.397,Z 454.962,A -85,B 0,C 180,E1 -20396.356,E2 -20396.356} C_VEL
LIN {X 0,Y 241.33,Z 466.232,A -85,B 0,C 180,E1 -20397.501,E2 -20397.501} C_VEL
LIN {X 0,Y 238.784,Z 477.647,A -85,B 0,C 180,E1 -20398.998,E2 -20398.998} C_VEL
LIN {X 0,Y 235.752,Z 488.437,A -85,B 0,C 180,E1 -20400.781,E2 -20400.781} C_VEL
LIN {X 0,Y 232.403,Z 499.089,A -85,B 0,C 180,E1 -20403.025,E2 -20403.025} C_VEL
LIN {X 0,Y 229.204,Z 508.47,A -85,B 0,C 180,E1 -20405.547,E2 -20405.547} C_VEL
LIN {X 0,Y 226.396,Z 516.025,A -85,B 0,C 180,E1 -20408.13,E2 -20408.13} C_VEL
LIN {X 0,Y 224.149,Z 522.161,A -85,B 0,C 180,E1 -20410.779,E2 -20410.779} C_VEL
LIN {X 0,Y 222.307,Z 527.102,A -85,B 0,C 180,E1 -20413.47,E2 -20413.47} C_VEL
LIN {X 0,Y 220.786,Z 530.989,A -85,B 0,C 180,E1 -20416.188,E2 -20416.188} C_VEL
LIN {X 0,Y 219.813,Z 533.883,A -85,B 0,C 180,E1 -20418.94,E2 -20418.94} C_VEL
LIN {X 0,Y 219.298,Z 535.34,A -85,B 0,C 180,E1 -20420.779,E2 -20420.779} C_VEL
LIN {X 0,Y 218.699,Z 537.07,A -85,B 0,C 180,E1 -20424.468,E2 -20424.468} C_VEL
LIN {X 0,Y 218.635,Z 537.367,A -85,B 0,C 180,E1 -20428.158,E2 -20428.158} C_VEL
LIN {X 0,Y 218.771,Z 536.253,A -85,B 0,C 180,E1 -20431.841,E2 -20431.841} C_VEL
LIN {X 0,Y 219.365,Z 533.613,A -85,B 0,C 180,E1 -20435.515,E2 -20435.515} C_VEL
LIN {X 0,Y 220.44,Z 529.428,A -85,B 0,C 180,E1 -20439.172,E2 -20439.172} C_VEL
LIN {X 0,Y 221.651,Z 525.13,A -85,B 0,C 180,E1 -20441.893,E2 -20441.893} C_VEL
LIN {X 0,Y 223.644,Z 518.741,A -85,B 0,C 180,E1 -20445.026,E2 -20445.026} C_VEL
LIN {X 0,Y 225.832,Z 511.837,A -85,B 0,C 180,E1 -20447.663,E2 -20447.663} C_VEL
LIN {X 0,Y 228.418,Z 503.309,A -85,B 0,C 180,E1 -20450.251,E2 -20450.251} C_VEL
LIN {X 0,Y 230.86,Z 494.676,A -85,B 0,C 180,E1 -20452.366,E2 -20452.366} C_VEL
LIN {X 0,Y 233.626,Z 484.137,A -85,B 0,C 180,E1 -20454.433,E2 -20454.433} C_VEL
LIN {X 0,Y 236.059,Z 473.757,A -85,B 0,C 180,E1 -20456.048,E2 -20456.048} C_VEL
LIN {X 0,Y 238.31,Z 462.473,A -85,B 0,C 180,E1 -20457.438,E2 -20457.438} C_VEL
LIN {X 0,Y 240.281,Z 449.716,A -85,B 0,C 180,E1 -20458.637,E2 -20458.637} C_VEL
LIN {X 0,Y 241.8,Z 436.8,A -85,B 0,C 180,E1 -20459.486,E2 -20459.486} C_VEL
LIN {X 0,Y 242.785,Z 423.859,A -85,B 0,C 180,E1 -20460.031,E2 -20460.031} C_VEL
LIN {X 0,Y 245.277,Z 361.947,A -85,B 0,C 180,E1 -20461.709,E2 -20461.709} C_VEL
LIN {X 0,Y 241.237,Z 334.404,A -85,B 0,C 180,E1 -20463.298,E2 -20463.298} C_VEL
LIN {X 0,Y 235.042,Z 320.823,A -85,B 0,C 180,E1 -20464.883,E2 -20464.883} C_VEL
LIN {X 0,Y 229.074,Z 308.862,A -85,B 0,C 180,E1 -20466.554,E2 -20466.554} C_VEL
LIN {X 0,Y 227.415,Z 302.27,A -85,B 0,C 180,E1 -20469.411,E2 -20469.411} C_VEL
LIN {X 0,Y 225.107,Z 294.103,A -85,B 0,C 180,E1 -20473.38,E2 -20473.38} C_VEL
LIN {X 0,Y 222.564,Z 286.123,A -85,B 0,C 180,E1 -20477.725,E2 -20477.725} C_VEL
LIN {X 0,Y 220.823,Z 280.676,A -85,B 0,C 180,E1 -20481.055,E2 -20481.055} C_VEL
LIN {X 0,Y 220.819,Z 280.564,A -85,B 0,C 180,E1 -20485.841,E2 -20485.841} C_VEL
LIN {X 0,Y 220.867,Z 280.596,A -85,B 0,C 180,E1 -20489.394,E2 -20489.394} C_VEL
LIN {X 0,Y 220.893,Z 280.596,A -85,B 0,C 180,E1 -20493.548,E2 -20493.548} C_VEL
LIN {X 0,Y 220.876,Z 280.595,A -85,B 0,C 180,E1 -20497.552,E2 -20497.552} C_VEL
LIN {X 0,Y 220.982,Z 280.584,A -85,B 0,C 180,E1 -20502.57,E2 -20502.57} C_VEL
LIN {X 0,Y 221.007,Z 280.58,A -85,B 0,C 180,E1 -20507.138,E2 -20507.138} C_VEL
LIN {X 0,Y 221.201,Z 280.541,A -85,B 0,C 180,E1 -20510.859,E2 -20510.859} C_VEL
LIN {X 0,Y 221.268,Z 280.55,A -85,B 0,C 180,E1 -20512.7,E2 -20512.7} C_VEL
LIN {X 0,Y 221.508,Z 280.52,A -85,B 0,C 180,E1 -20518.181,E2 -20518.181} C_VEL
LIN {X 0,Y 221.509,Z 280.506,A -85,B 0,C 180,E1 -20521.818,E2 -20521.818} C_VEL
LIN {X 0,Y 221.286,Z 280.535,A -85,B 0,C 180,E1 -20527.298,E2 -20527.298} C_VEL
LIN {X 0,Y 221.103,Z 280.551,A -85,B 0,C 180,E1 -20530.994,E2 -20530.994} C_VEL
LIN {X 0,Y 221.012,Z 280.567,A -85,B 0,C 180,E1 -20536.63,E2 -20536.63} C_VEL
LIN {X 0,Y 220.889,Z 280.582,A -85,B 0,C 180,E1 -20540.486,E2 -20540.486} C_VEL
LIN {X 0,Y 220.863,Z 280.587,A -85,B 0,C 180,E1 -20544.435,E2 -20544.435} C_VEL
LIN {X 0,Y 220.827,Z 280.584,A -85,B 0,C 180,E1 -20547.948,E2 -20547.948} C_VEL
LIN {X 0,Y 220.127,Z 280.657,A -85,B 0,C 180,E1 -20548.959,E2 -20548.959} C_VEL
LIN {X 0,Y 217.257,Z 281.007,A -85,B 0,C 180,E1 -20550.546,E2 -20550.546} C_VEL
LIN {X 0,Y 214.385,Z 281.376,A -85,B 0,C 180,E1 -20552.173,E2 -20552.173} C_VEL
LIN {X 0,Y 213.724,Z 281.472,A -85,B 0,C 180,E1 -20553.23,E2 -20553.23} C_VEL
LIN {X 0,Y 213.789,Z 281.699,A -85,B 0,C 180,E1 -20555.194,E2 -20555.194} C_VEL
LIN {X 0,Y 216.085,Z 288.328,A -85,B 0,C 180,E1 -20559.36,E2 -20559.36} C_VEL
LIN {X 0,Y 218.639,Z 296.22,A -85,B 0,C 180,E1 -20563.717,E2 -20563.717} C_VEL
LIN {X 0,Y 220.469,Z 302.309,A -85,B 0,C 180,E1 -20566.652,E2 -20566.652} C_VEL
LIN {X 0,Y 227.946,Z 315.623,A -85,B 0,C 180,E1 -20568.86,E2 -20568.86} C_VEL
LIN {X 0,Y 234.506,Z 328.783,A -85,B 0,C 180,E1 -20570.646,E2 -20570.646} C_VEL
LIN {X 0,Y 240.58,Z 342.836,A -85,B 0,C 180,E1 -20572.257,E2 -20572.257} C_VEL
LIN {X 0,Y 240.505,Z 348.913,A -85,B 0,C 180,E1 -20572.471,E2 -20572.471} C_VEL
LIN {X 0,Y 236.488,Z 429.789,A -85,B 0,C 180,E1 -20574.846,E2 -20574.846} C_VEL
LIN {X 0,Y 235.193,Z 443.598,A -85,B 0,C 180,E1 -20575.537,E2 -20575.537} C_VEL
LIN {X 0,Y 233.446,Z 455.876,A -85,B 0,C 180,E1 -20576.415,E2 -20576.415} C_VEL
LIN {X 0,Y 231.282,Z 468.252,A -85,B 0,C 180,E1 -20577.618,E2 -20577.618} C_VEL
LIN {X 0,Y 228.807,Z 480.291,A -85,B 0,C 180,E1 -20579.144,E2 -20579.144} C_VEL
LIN {X 0,Y 225.826,Z 492.747,A -85,B 0,C 180,E1 -20581.16,E2 -20581.16} C_VEL
LIN {X 0,Y 222.912,Z 503.315,A -85,B 0,C 180,E1 -20583.303,E2 -20583.303} C_VEL
LIN {X 0,Y 220.381,Z 512.102,A -85,B 0,C 180,E1 -20585.508,E2 -20585.508} C_VEL
LIN {X 0,Y 217.784,Z 520.911,A -85,B 0,C 180,E1 -20588.216,E2 -20588.216} C_VEL
LIN {X 0,Y 215.523,Z 529.237,A -85,B 0,C 180,E1 -20591.462,E2 -20591.462} C_VEL
LIN {X 0,Y 213.671,Z 535.852,A -85,B 0,C 180,E1 -20594.744,E2 -20594.744} C_VEL
LIN {X 0,Y 212.504,Z 540.379,A -85,B 0,C 180,E1 -20597.587,E2 -20597.587} C_VEL
LIN {X 0,Y 211.876,Z 543.924,A -85,B 0,C 180,E1 -20600.454,E2 -20600.454} C_VEL
LIN {X 0,Y 211.595,Z 545.788,A -85,B 0,C 180,E1 -20602.365,E2 -20602.365} C_VEL
LIN {X 0,Y 211.349,Z 548.335,A -85,B 0,C 180,E1 -20606.187,E2 -20606.187} C_VEL
LIN {X 0,Y 211.43,Z 549.061,A -85,B 0,C 180,E1 -20608.095,E2 -20608.095} C_VEL
LIN {X 0,Y 211.545,Z 549.427,A -85,B 0,C 180,E1 -20610,E2 -20610} C_VEL
LIN {X 0,Y 211.415,Z 549.065,A -85,B 0,C 180,E1 -20613.812,E2 -20613.812} C_VEL
LIN {X 0,Y 211.609,Z 547.268,A -85,B 0,C 180,E1 -20617.634,E2 -20617.634} C_VEL
LIN {X 0,Y 212.331,Z 543.987,A -85,B 0,C 180,E1 -20621.455,E2 -20621.455} C_VEL
LIN {X 0,Y 213.807,Z 539.081,A -85,B 0,C 180,E1 -20625.246,E2 -20625.246} C_VEL
LIN {X 0,Y 215.443,Z 534.298,A -85,B 0,C 180,E1 -20628.053,E2 -20628.053} C_VEL
LIN {X 0,Y 217.749,Z 527.286,A -85,B 0,C 180,E1 -20631.29,E2 -20631.29} C_VEL
LIN {X 0,Y 220.815,Z 518.528,A -85,B 0,C 180,E1 -20634.441,E2 -20634.441} C_VEL
LIN {X 0,Y 223.954,Z 509.302,A -85,B 0,C 180,E1 -20637.066,E2 -20637.066} C_VEL
LIN {X 0,Y 227.356,Z 499.019,A -85,B 0,C 180,E1 -20639.388,E2 -20639.388} C_VEL
LIN {X 0,Y 230.55,Z 487.54,A -85,B 0,C 180,E1 -20641.468,E2 -20641.468} C_VEL
LIN {X 0,Y 233.76,Z 474.723,A -85,B 0,C 180,E1 -20643.276,E2 -20643.276} C_VEL
LIN {X 0,Y 236.631,Z 461.09,A -85,B 0,C 180,E1 -20644.741,E2 -20644.741} C_VEL
LIN {X 0,Y 238.877,Z 447.694,A -85,B 0,C 180,E1 -20645.784,E2 -20645.784} C_VEL
LIN {X 0,Y 240.563,Z 433.783,A -85,B 0,C 180,E1 -20646.53,E2 -20646.53} C_VEL
LIN {X 0,Y 241.878,Z 414.556,A -85,B 0,C 180,E1 -20647.143,E2 -20647.143} C_VEL
LIN {X 0,Y 245.166,Z 348.069,A -85,B 0,C 180,E1 -20649.064,E2 -20649.064} C_VEL
LIN {X 0,Y 237.851,Z 331.923,A -85,B 0,C 180,E1 -20651.141,E2 -20651.141} C_VEL
LIN {X 0,Y 229.352,Z 316.078,A -85,B 0,C 180,E1 -20653.677,E2 -20653.677} C_VEL
LIN {X 0,Y 223.214,Z 306.272,A -85,B 0,C 180,E1 -20655.628,E2 -20655.628} C_VEL
LIN {X 0,Y 220.881,Z 302.279,A -85,B 0,C 180,E1 -20656.524,E2 -20656.524} C_VEL
LIN {X 0,Y 218.588,Z 295.194,A -85,B 0,C 180,E1 -20660.501,E2 -20660.501} C_VEL
LIN {X 0,Y 216.135,Z 287.944,A -85,B 0,C 180,E1 -20665.163,E2 -20665.163} C_VEL
LIN {X 0,Y 213.793,Z 281.61,A -85,B 0,C 180,E1 -20670.071,E2 -20670.071} C_VEL
LIN {X 0,Y 213.823,Z 281.455,A -85,B 0,C 180,E1 -20672.603,E2 -20672.603} C_VEL
LIN {X 0,Y 213.849,Z 281.468,A -85,B 0,C 180,E1 -20676.953,E2 -20676.953} C_VEL
LIN {X 0,Y 213.941,Z 281.45,A -85,B 0,C 180,E1 -20682.804,E2 -20682.804} C_VEL
LIN {X 0,Y 213.951,Z 281.452,A -85,B 0,C 180,E1 -20686.707,E2 -20686.707} C_VEL
LIN {X 0,Y 214.164,Z 281.433,A -85,B 0,C 180,E1 -20690.557,E2 -20690.557} C_VEL
LIN {X 0,Y 214.223,Z 281.409,A -85,B 0,C 180,E1 -20692.46,E2 -20692.46} C_VEL
LIN {X 0,Y 214.442,Z 281.383,A -85,B 0,C 180,E1 -20698.123,E2 -20698.123} C_VEL
LIN {X 0,Y 214.547,Z 281.386,A -85,B 0,C 180,E1 -20700.001,E2 -20700.001} C_VEL
LIN {X 0,Y 214.443,Z 281.382,A -85,B 0,C 180,E1 -20701.879,E2 -20701.879} C_VEL
LIN {X 0,Y 214.225,Z 281.41,A -85,B 0,C 180,E1 -20707.541,E2 -20707.541} C_VEL
LIN {X 0,Y 214.021,Z 281.435,A -85,B 0,C 180,E1 -20711.364,E2 -20711.364} C_VEL
LIN {X 0,Y 213.93,Z 281.449,A -85,B 0,C 180,E1 -20715.238,E2 -20715.238} C_VEL
LIN {X 0,Y 213.84,Z 281.463,A -85,B 0,C 180,E1 -20719.188,E2 -20719.188} C_VEL
LIN {X 0,Y 213.853,Z 281.463,A -85,B 0,C 180,E1 -20723.227,E2 -20723.227} C_VEL
LIN {X 0,Y 213.822,Z 281.618,A -85,B 0,C 180,E1 -20727.936,E2 -20727.936} C_VEL
LIN {X 0,Y 215.925,Z 287.34,A -85,B 0,C 180,E1 -20732.483,E2 -20732.483} C_VEL
LIN {X 0,Y 217.993,Z 293.433,A -85,B 0,C 180,E1 -20736.615,E2 -20736.615} C_VEL
LIN {X 0,Y 220.123,Z 300.628,A -85,B 0,C 180,E1 -20740.883,E2 -20740.883} C_VEL
LIN {X 0,Y 222.35,Z 308.405,A -85,B 0,C 180,E1 -20744.962,E2 -20744.962} C_VEL
LIN {X 0,Y 225.163,Z 313.308,A -85,B 0,C 180,E1 -20745.961,E2 -20745.961} C_VEL
LIN {X 0,Y 233.211,Z 327.977,A -85,B 0,C 180,E1 -20748.46,E2 -20748.46} C_VEL
LIN {X 0,Y 238.863,Z 339.812,A -85,B 0,C 180,E1 -20750.106,E2 -20750.106} C_VEL
LIN {X 0,Y 240.893,Z 344.61,A -85,B 0,C 180,E1 -20750.687,E2 -20750.687} C_VEL
LIN {X 0,Y 244.016,Z 366.093,A -85,B 0,C 180,E1 -20752.051,E2 -20752.051} C_VEL
LIN {X 0,Y 241.109,Z 427.133,A -85,B 0,C 180,E1 -20753.707,E2 -20753.707} C_VEL
LIN {X 0,Y 239.674,Z 440.788,A -85,B 0,C 180,E1 -20754.353,E2 -20754.353} C_VEL
LIN {X 0,Y 237.714,Z 453.924,A -85,B 0,C 180,E1 -20755.311,E2 -20755.311} C_VEL
LIN {X 0,Y 235.384,Z 466.327,A -85,B 0,C 180,E1 -20756.574,E2 -20756.574} C_VEL
LIN {X 0,Y 232.657,Z 478.033,A -85,B 0,C 180,E1 -20758.144,E2 -20758.144} C_VEL
LIN {X 0,Y 229.591,Z 488.541,A -85,B 0,C 180,E1 -20759.918,E2 -20759.918} C_VEL
LIN {X 0,Y 226.071,Z 499.202,A -85,B 0,C 180,E1 -20762.205,E2 -20762.205} C_VEL
LIN {X 0,Y 222.755,Z 508.592,A -85,B 0,C 180,E1 -20764.791,E2 -20764.791} C_VEL
LIN {X 0,Y 219.797,Z 516.158,A -85,B 0,C 180,E1 -20767.437,E2 -20767.437} C_VEL
LIN {X 0,Y 217.43,Z 522.304,A -85,B 0,C 180,E1 -20770.16,E2 -20770.16} C_VEL
LIN {X 0,Y 215.483,Z 527.255,A -85,B 0,C 180,E1 -20772.93,E2 -20772.93} C_VEL
LIN {X 0,Y 213.871,Z 531.149,A -85,B 0,C 180,E1 -20775.732,E2 -20775.732} C_VEL
LIN {X 0,Y 212.812,Z 534.052,A -85,B 0,C 180,E1 -20778.571,E2 -20778.571} C_VEL
LIN {X 0,Y 212.268,Z 535.517,A -85,B 0,C 180,E1 -20780.471,E2 -20780.471} C_VEL
LIN {X 0,Y 211.641,Z 537.26,A -85,B 0,C 180,E1 -20784.283,E2 -20784.283} C_VEL
LIN {X 0,Y 211.534,Z 537.569,A -85,B 0,C 180,E1 -20788.096,E2 -20788.096} C_VEL
LIN {X 0,Y 211.692,Z 536.468,A -85,B 0,C 180,E1 -20791.902,E2 -20791.902} C_VEL
LIN {X 0,Y 211.95,Z 535.348,A -85,B 0,C 180,E1 -20793.802,E2 -20793.802} C_VEL
LIN {X 0,Y 212.777,Z 531.962,A -85,B 0,C 180,E1 -20797.592,E2 -20797.592} C_VEL
LIN {X 0,Y 213.82,Z 528.36,A -85,B 0,C 180,E1 -20800.415,E2 -20800.415} C_VEL
LIN {X 0,Y 215.253,Z 523.737,A -85,B 0,C 180,E1 -20803.211,E2 -20803.211} C_VEL
LIN {X 0,Y 217.539,Z 516.863,A -85,B 0,C 180,E1 -20806.42,E2 -20806.42} C_VEL
LIN {X 0,Y 219.937,Z 509.497,A -85,B 0,C 180,E1 -20809.119,E2 -20809.119} C_VEL
LIN {X 0,Y 222.763,Z 500.441,A -85,B 0,C 180,E1 -20811.759,E2 -20811.759} C_VEL
LIN {X 0,Y 225.715,Z 490.101,A -85,B 0,C 180,E1 -20814.121,E2 -20814.121} C_VEL
LIN {X 0,Y 228.363,Z 479.693,A -85,B 0,C 180,E1 -20816.011,E2 -20816.011} C_VEL
LIN {X 0,Y 231.027,Z 468.211,A -85,B 0,C 180,E1 -20817.639,E2 -20817.639} C_VEL
LIN {X 0,Y 233.266,Z 456.432,A -85,B 0,C 180,E1 -20818.932,E2 -20818.932} C_VEL
LIN {X 0,Y 234.94,Z 443.939,A -85,B 0,C 180,E1 -20819.97,E2 -20819.97} C_VEL
LIN {X 0,Y 236.394,Z 430.402,A -85,B 0,C 180,E1 -20820.703,E2 -20820.703} C_VEL
LIN {X 0,Y 237.332,Z 412.874,A -85,B 0,C 180,E1 -20821.258,E2 -20821.258} C_VEL
LIN {X 0,Y 239.314,Z 362.022,A -85,B 0,C 180,E1 -20822.677,E2 -20822.677} C_VEL
LIN {X 0,Y 235.624,Z 336.96,A -85,B 0,C 180,E1 -20824.192,E2 -20824.192} C_VEL
LIN {X 0,Y 228.647,Z 321.704,A -85,B 0,C 180,E1 -20826.079,E2 -20826.079} C_VEL
LIN {X 0,Y 223.248,Z 311.542,A -85,B 0,C 180,E1 -20827.593,E2 -20827.593} C_VEL
LIN {X 0,Y 221.818,Z 308.438,A -85,B 0,C 180,E1 -20828.149,E2 -20828.149} C_VEL
LIN {X 0,Y 219.55,Z 299.87,A -85,B 0,C 180,E1 -20832.238,E2 -20832.238} C_VEL
LIN {X 0,Y 217.496,Z 293.038,A -85,B 0,C 180,E1 -20835.891,E2 -20835.891} C_VEL
LIN {X 0,Y 215.652,Z 287.176,A -85,B 0,C 180,E1 -20839.322,E2 -20839.322} C_VEL
LIN {X 0,Y 213.78,Z 281.562,A -85,B 0,C 180,E1 -20843.031,E2 -20843.031} C_VEL
LIN {X 0,Y 213.767,Z 281.441,A -85,B 0,C 180,E1 -20846.019,E2 -20846.019} C_VEL
LIN {X 0,Y 213.779,Z 281.476,A -85,B 0,C 180,E1 -20850.453,E2 -20850.453} C_VEL
LIN {X 0,Y 213.8,Z 281.47,A -85,B 0,C 180,E1 -20854.701,E2 -20854.701} C_VEL
LIN {X 0,Y 213.811,Z 281.472,A -85,B 0,C 180,E1 -20858.802,E2 -20858.802} C_VEL
LIN {X 0,Y 213.941,Z 281.461,A -85,B 0,C 180,E1 -20862.803,E2 -20862.803} C_VEL
LIN {X 0,Y 213.949,Z 281.454,A -85,B 0,C 180,E1 -20866.706,E2 -20866.706} C_VEL
LIN {X 0,Y 214.139,Z 281.419,A -85,B 0,C 180,E1 -20870.554,E2 -20870.554} C_VEL
LIN {X 0,Y 214.205,Z 281.428,A -85,B 0,C 180,E1 -20872.458,E2 -20872.458} C_VEL
LIN {X 0,Y 214.441,Z 281.4,A -85,B 0,C 180,E1 -20878.121,E2 -20878.121} C_VEL
LIN {X 0,Y 214.546,Z 281.369,A -85,B 0,C 180,E1 -20879.999,E2 -20879.999} C_VEL
LIN {X 0,Y 214.442,Z 281.386,A -85,B 0,C 180,E1 -20881.877,E2 -20881.877} C_VEL
LIN {X 0,Y 214.224,Z 281.417,A -85,B 0,C 180,E1 -20887.54,E2 -20887.54} C_VEL
LIN {X 0,Y 214.019,Z 281.434,A -85,B 0,C 180,E1 -20891.363,E2 -20891.363} C_VEL
LIN {X 0,Y 213.928,Z 281.449,A -85,B 0,C 180,E1 -20895.237,E2 -20895.237} C_VEL
LIN {X 0,Y 213.836,Z 281.468,A -85,B 0,C 180,E1 -20899.187,E2 -20899.187} C_VEL
LIN {X 0,Y 213.844,Z 281.47,A -85,B 0,C 180,E1 -20903.227,E2 -20903.227} C_VEL
LIN {X 0,Y 213.786,Z 281.462,A -85,B 0,C 180,E1 -20907.914,E2 -20907.914} C_VEL
LIN {X 0,Y 213.765,Z 281.447,A -85,B 0,C 180,E1 -20911.737,E2 -20911.737} C_VEL
LIN {X 0,Y 213.724,Z 281.472,A -85,B 0,C 180,E1 -20913.23,E2 -20913.23} C_VEL
LIN {X 0,Y 213.553,Z 281.935,A -85,B 0,C 180,E1 -20914.27,E2 -20914.27} C_VEL
LIN {X 0,Y 212.804,Z 283.883,A -85,B 0,C 180,E1 -20915.758,E2 -20915.758} C_VEL
LIN {X 0,Y 211.823,Z 286.701,A -85,B 0,C 180,E1 -20917.16,E2 -20917.16} C_VEL
LIN {X 0,Y 210.769,Z 291.062,A -85,B 0,C 180,E1 -20919.019,E2 -20919.019} C_VEL
LIN {X 0,Y 210.723,Z 294.015,A -85,B 0,C 180,E1 -20920.452,E2 -20920.452} C_VEL
LIN {X 0,Y 210.936,Z 294.893,A -85,B 0,C 180,E1 -20920.941,E2 -20920.941} C_VEL
LIN {X 0,Y 213.29,Z 302.405,A -85,B 0,C 180,E1 -20924.94,E2 -20924.94} C_VEL
LIN {X 0,Y 218.86,Z 312.003,A -85,B 0,C 180,E1 -20926.763,E2 -20926.763} C_VEL
LIN {X 0,Y 225.865,Z 325.01,A -85,B 0,C 180,E1 -20928.813,E2 -20928.813} C_VEL
LIN {X 0,Y 232.833,Z 340.235,A -85,B 0,C 180,E1 -20930.783,E2 -20930.783} C_VEL
LIN {X 0,Y 234.856,Z 345.22,A -85,B 0,C 180,E1 -20931.346,E2 -20931.346} C_VEL
LIN {X 0,Y 230.594,Z 429.497,A -85,B 0,C 180,E1 -20933.875,E2 -20933.875} C_VEL
LIN {X 0,Y 229.253,Z 443.413,A -85,B 0,C 180,E1 -20934.579,E2 -20934.579} C_VEL
LIN {X 0,Y 227.349,Z 456.287,A -85,B 0,C 180,E1 -20935.523,E2 -20935.523} C_VEL
LIN {X 0,Y 224.939,Z 469.444,A -85,B 0,C 180,E1 -20936.855,E2 -20936.855} C_VEL
LIN {X 0,Y 222.311,Z 481.507,A -85,B 0,C 180,E1 -20938.455,E2 -20938.455} C_VEL
LIN {X 0,Y 219.294,Z 493.504,A -85,B 0,C 180,E1 -20940.48,E2 -20940.48} C_VEL
LIN {X 0,Y 216.554,Z 502.934,A -85,B 0,C 180,E1 -20942.454,E2 -20942.454} C_VEL
LIN {X 0,Y 213.88,Z 511.757,A -85,B 0,C 180,E1 -20944.712,E2 -20944.712} C_VEL
LIN {X 0,Y 211.143,Z 520.596,A -85,B 0,C 180,E1 -20947.494,E2 -20947.494} C_VEL
LIN {X 0,Y 208.755,Z 528.714,A -85,B 0,C 180,E1 -20950.719,E2 -20950.719} C_VEL
LIN {X 0,Y 207.272,Z 533.854,A -85,B 0,C 180,E1 -20953.25,E2 -20953.25} C_VEL
LIN {X 0,Y 205.861,Z 538.715,A -85,B 0,C 180,E1 -20956.174,E2 -20956.174} C_VEL
LIN {X 0,Y 204.836,Z 543.685,A -85,B 0,C 180,E1 -20960.122,E2 -20960.122} C_VEL
LIN {X 0,Y 204.532,Z 545.56,A -85,B 0,C 180,E1 -20962.1,E2 -20962.1} C_VEL
LIN {X 0,Y 204.258,Z 548.122,A -85,B 0,C 180,E1 -20966.054,E2 -20966.054} C_VEL
LIN {X 0,Y 204.331,Z 548.854,A -85,B 0,C 180,E1 -20968.029,E2 -20968.029} C_VEL
LIN {X 0,Y 204.462,Z 549.226,A -85,B 0,C 180,E1 -20970,E2 -20970} C_VEL
LIN {X 0,Y 204.335,Z 548.873,A -85,B 0,C 180,E1 -20973.944,E2 -20973.944} C_VEL
LIN {X 0,Y 204.545,Z 547.086,A -85,B 0,C 180,E1 -20977.9,E2 -20977.9} C_VEL
LIN {X 0,Y 205.34,Z 543.818,A -85,B 0,C 180,E1 -20981.85,E2 -20981.85} C_VEL
LIN {X 0,Y 206.433,Z 540.303,A -85,B 0,C 180,E1 -20984.793,E2 -20984.793} C_VEL
LIN {X 0,Y 207.999,Z 535.838,A -85,B 0,C 180,E1 -20987.704,E2 -20987.704} C_VEL
LIN {X 0,Y 210.307,Z 529.365,A -85,B 0,C 180,E1 -20991.025,E2 -20991.025} C_VEL
LIN {X 0,Y 212.872,Z 522.381,A -85,B 0,C 180,E1 -20993.855,E2 -20993.855} C_VEL
LIN {X 0,Y 215.914,Z 514.004,A -85,B 0,C 180,E1 -20996.587,E2 -20996.587} C_VEL
LIN {X 0,Y 219.536,Z 503.826,A -85,B 0,C 180,E1 -20999.222,E2 -20999.222} C_VEL
LIN {X 0,Y 222.87,Z 493.289,A -85,B 0,C 180,E1 -21001.39,E2 -21001.39} C_VEL
LIN {X 0,Y 225.976,Z 482.09,A -85,B 0,C 180,E1 -21003.239,E2 -21003.239} C_VEL
LIN {X 0,Y 229.001,Z 469.543,A -85,B 0,C 180,E1 -21004.861,E2 -21004.861} C_VEL
LIN {X 0,Y 231.687,Z 456.486,A -85,B 0,C 180,E1 -21006.129,E2 -21006.129} C_VEL
LIN {X 0,Y 233.845,Z 443,A -85,B 0,C 180,E1 -21007.082,E2 -21007.082} C_VEL
LIN {X 0,Y 235.33,Z 428.852,A -85,B 0,C 180,E1 -21007.75,E2 -21007.75} C_VEL
LIN {X 0,Y 239.536,Z 350.249,A -85,B 0,C 180,E1 -21010.064,E2 -21010.064} C_VEL
LIN {X 0,Y 232.835,Z 335.364,A -85,B 0,C 180,E1 -21012.069,E2 -21012.069} C_VEL
LIN {X 0,Y 224.932,Z 320.508,A -85,B 0,C 180,E1 -21014.547,E2 -21014.547} C_VEL
LIN {X 0,Y 219.171,Z 311.152,A -85,B 0,C 180,E1 -21016.469,E2 -21016.469} C_VEL
LIN {X 0,Y 215.822,Z 306.061,A -85,B 0,C 180,E1 -21017.65,E2 -21017.65} C_VEL
LIN {X 0,Y 213.714,Z 302.44,A -85,B 0,C 180,E1 -21018.562,E2 -21018.562} C_VEL
LIN {X 0,Y 211.359,Z 295.323,A -85,B 0,C 180,E1 -21022.942,E2 -21022.942} C_VEL
LIN {X 0,Y 209.626,Z 290.379,A -85,B 0,C 180,E1 -21026.416,E2 -21026.416} C_VEL
LIN {X 0,Y 207.707,Z 285.191,A -85,B 0,C 180,E1 -21030.619,E2 -21030.619} C_VEL
LIN {X 0,Y 206.757,Z 282.406,A -85,B 0,C 180,E1 -21033.305,E2 -21033.305} C_VEL
LIN {X 0,Y 206.759,Z 282.351,A -85,B 0,C 180,E1 -21038.044,E2 -21038.044} C_VEL
LIN {X 0,Y 206.871,Z 282.336,A -85,B 0,C 180,E1 -21042.197,E2 -21042.197} C_VEL
LIN {X 0,Y 206.893,Z 282.336,A -85,B 0,C 180,E1 -21046.245,E2 -21046.245} C_VEL
LIN {X 0,Y 207.103,Z 282.312,A -85,B 0,C 180,E1 -21050.232,E2 -21050.232} C_VEL
LIN {X 0,Y 207.164,Z 282.289,A -85,B 0,C 180,E1 -21052.202,E2 -21052.202} C_VEL
LIN {X 0,Y 207.379,Z 282.263,A -85,B 0,C 180,E1 -21058.059,E2 -21058.059} C_VEL
LIN {X 0,Y 207.512,Z 282.262,A -85,B 0,C 180,E1 -21060.001,E2 -21060.001} C_VEL
LIN {X 0,Y 207.38,Z 282.262,A -85,B 0,C 180,E1 -21061.943,E2 -21061.943} C_VEL
LIN {X 0,Y 207.166,Z 282.291,A -85,B 0,C 180,E1 -21067.8,E2 -21067.8} C_VEL
LIN {X 0,Y 206.941,Z 282.317,A -85,B 0,C 180,E1 -21071.758,E2 -21071.758} C_VEL
LIN {X 0,Y 206.863,Z 282.328,A -85,B 0,C 180,E1 -21075.772,E2 -21075.772} C_VEL
LIN {X 0,Y 206.79,Z 282.339,A -85,B 0,C 180,E1 -21079.869,E2 -21079.869} C_VEL
LIN {X 0,Y 206.764,Z 282.458,A -85,B 0,C 180,E1 -21084.808,E2 -21084.808} C_VEL
LIN {X 0,Y 208.24,Z 286.618,A -85,B 0,C 180,E1 -21088.661,E2 -21088.661} C_VEL
LIN {X 0,Y 210.001,Z 291.262,A -85,B 0,C 180,E1 -21092.376,E2 -21092.376} C_VEL
LIN {X 0,Y 212.022,Z 297.356,A -85,B 0,C 180,E1 -21096.632,E2 -21096.632} C_VEL
LIN {X 0,Y 214.102,Z 304.629,A -85,B 0,C 180,E1 -21101.035,E2 -21101.035} C_VEL
LIN {X 0,Y 215.246,Z 308.418,A -85,B 0,C 180,E1 -21103.049,E2 -21103.049} C_VEL
LIN {X 0,Y 219.399,Z 315.535,A -85,B 0,C 180,E1 -21104.57,E2 -21104.57} C_VEL
LIN {X 0,Y 224.267,Z 323.893,A -85,B 0,C 180,E1 -21106.199,E2 -21106.199} C_VEL
LIN {X 0,Y 230.998,Z 336.914,A -85,B 0,C 180,E1 -21108.324,E2 -21108.324} C_VEL
LIN {X 0,Y 235.694,Z 347.6,A -85,B 0,C 180,E1 -21109.747,E2 -21109.747} C_VEL
LIN {X 0,Y 238.434,Z 366.69,A -85,B 0,C 180,E1 -21111.009,E2 -21111.009} C_VEL
LIN {X 0,Y 235.402,Z 427.749,A -85,B 0,C 180,E1 -21112.706,E2 -21112.706} C_VEL
LIN {X 0,Y 233.956,Z 440.894,A -85,B 0,C 180,E1 -21113.342,E2 -21113.342} C_VEL
LIN {X 0,Y 231.911,Z 454.02,A -85,B 0,C 180,E1 -21114.313,E2 -21114.313} C_VEL
LIN {X 0,Y 229.481,Z 466.421,A -85,B 0,C 180,E1 -21115.595,E2 -21115.595} C_VEL
LIN {X 0,Y 226.573,Z 478.438,A -85,B 0,C 180,E1 -21117.246,E2 -21117.246} C_VEL
LIN {X 0,Y 223.115,Z 489.708,A -85,B 0,C 180,E1 -21119.212,E2 -21119.212} C_VEL
LIN {X 0,Y 219.794,Z 499.314,A -85,B 0,C 180,E1 -21121.339,E2 -21121.339} C_VEL
LIN {X 0,Y 216.342,Z 508.714,A -85,B 0,C 180,E1 -21123.989,E2 -21123.989} C_VEL
LIN {X 0,Y 213.227,Z 516.291,A -85,B 0,C 180,E1 -21126.702,E2 -21126.702} C_VEL
LIN {X 0,Y 210.736,Z 522.447,A -85,B 0,C 180,E1 -21129.502,E2 -21129.502} C_VEL
LIN {X 0,Y 208.684,Z 527.407,A -85,B 0,C 180,E1 -21132.356,E2 -21132.356} C_VEL
LIN {X 0,Y 206.951,Z 531.31,A -85,B 0,C 180,E1 -21135.244,E2 -21135.244} C_VEL
LIN {X 0,Y 205.83,Z 534.221,A -85,B 0,C 180,E1 -21138.178,E2 -21138.178} C_VEL
LIN {X 0,Y 205.257,Z 535.693,A -85,B 0,C 180,E1 -21140.142,E2 -21140.142} C_VEL
LIN {X 0,Y 204.576,Z 537.45,A -85,B 0,C 180,E1 -21144.084,E2 -21144.084} C_VEL
LIN {X 0,Y 204.435,Z 537.771,A -85,B 0,C 180,E1 -21148.03,E2 -21148.03} C_VEL
LIN {X 0,Y 204.616,Z 536.683,A -85,B 0,C 180,E1 -21151.968,E2 -21151.968} C_VEL
LIN {X 0,Y 204.886,Z 535.574,A -85,B 0,C 180,E1 -21153.934,E2 -21153.934} C_VEL
LIN {X 0,Y 205.745,Z 532.202,A -85,B 0,C 180,E1 -21157.853,E2 -21157.853} C_VEL
LIN {X 0,Y 206.838,Z 528.616,A -85,B 0,C 180,E1 -21160.77,E2 -21160.77} C_VEL
LIN {X 0,Y 208.347,Z 524.012,A -85,B 0,C 180,E1 -21163.658,E2 -21163.658} C_VEL
LIN {X 0,Y 210.752,Z 517.157,A -85,B 0,C 180,E1 -21166.965,E2 -21166.965} C_VEL
LIN {X 0,Y 213.241,Z 509.818,A -85,B 0,C 180,E1 -21169.744,E2 -21169.744} C_VEL
LIN {X 0,Y 216.177,Z 500.803,A -85,B 0,C 180,E1 -21172.457,E2 -21172.457} C_VEL
LIN {X 0,Y 219.273,Z 490.518,A -85,B 0,C 180,E1 -21174.877,E2 -21174.877} C_VEL
LIN {X 0,Y 222.027,Z 480.17,A -85,B 0,C 180,E1 -21176.811,E2 -21176.811} C_VEL
LIN {X 0,Y 224.786,Z 468.77,A -85,B 0,C 180,E1 -21178.476,E2 -21178.476} C_VEL
LIN {X 0,Y 227.129,Z 457.023,A -85,B 0,C 180,E1 -21179.802,E2 -21179.802} C_VEL
LIN {X 0,Y 228.842,Z 445.173,A -85,B 0,C 180,E1 -21180.829,E2 -21180.829} C_VEL
LIN {X 0,Y 230.356,Z 431.855,A -85,B 0,C 180,E1 -21181.601,E2 -21181.601} C_VEL
LIN {X 0,Y 231.364,Z 415.04,A -85,B 0,C 180,E1 -21182.167,E2 -21182.167} C_VEL
LIN {X 0,Y 233.509,Z 363.119,A -85,B 0,C 180,E1 -21183.643,E2 -21183.643} C_VEL
LIN {X 0,Y 230.172,Z 339.763,A -85,B 0,C 180,E1 -21185.101,E2 -21185.101} C_VEL
LIN {X 0,Y 223.248,Z 324.729,A -85,B 0,C 180,E1 -21187.069,E2 -21187.069} C_VEL
LIN {X 0,Y 216.928,Z 312.616,A -85,B 0,C 180,E1 -21188.962,E2 -21188.962} C_VEL
LIN {X 0,Y 214.664,Z 308.329,A -85,B 0,C 180,E1 -21189.792,E2 -21189.792} C_VEL
LIN {X 0,Y 212.398,Z 300.035,A -85,B 0,C 180,E1 -21194.015,E2 -21194.015} C_VEL
LIN {X 0,Y 210.248,Z 293.067,A -85,B 0,C 180,E1 -21198.044,E2 -21198.044} C_VEL
LIN {X 0,Y 207.976,Z 286.128,A -85,B 0,C 180,E1 -21202.535,E2 -21202.535} C_VEL
LIN {X 0,Y 206.766,Z 282.419,A -85,B 0,C 180,E1 -21205.295,E2 -21205.295} C_VEL
LIN {X 0,Y 206.723,Z 282.353,A -85,B 0,C 180,E1 -21209.338,E2 -21209.338} C_VEL
LIN {X 0,Y 206.732,Z 282.36,A -85,B 0,C 180,E1 -21213.771,E2 -21213.771} C_VEL
LIN {X 0,Y 206.757,Z 282.357,A -85,B 0,C 180,E1 -21218.042,E2 -21218.042} C_VEL
LIN {X 0,Y 206.871,Z 282.34,A -85,B 0,C 180,E1 -21222.196,E2 -21222.196} C_VEL
LIN {X 0,Y 206.891,Z 282.327,A -85,B 0,C 180,E1 -21226.243,E2 -21226.243} C_VEL
LIN {X 0,Y 207.097,Z 282.296,A -85,B 0,C 180,E1 -21230.23,E2 -21230.23} C_VEL
LIN {X 0,Y 207.062,Z 282.305,A -85,B 0,C 180,E1 -21234.155,E2 -21234.155} C_VEL
LIN {X 0,Y 207.378,Z 282.279,A -85,B 0,C 180,E1 -21238.057,E2 -21238.057} C_VEL
LIN {X 0,Y 207.511,Z 282.245,A -85,B 0,C 180,E1 -21239.999,E2 -21239.999} C_VEL
LIN {X 0,Y 207.379,Z 282.266,A -85,B 0,C 180,E1 -21241.941,E2 -21241.941} C_VEL
LIN {X 0,Y 207.164,Z 282.299,A -85,B 0,C 180,E1 -21247.798,E2 -21247.798} C_VEL
LIN {X 0,Y 206.939,Z 282.317,A -85,B 0,C 180,E1 -21251.757,E2 -21251.757} C_VEL
LIN {X 0,Y 206.861,Z 282.327,A -85,B 0,C 180,E1 -21255.771,E2 -21255.771} C_VEL
LIN {X 0,Y 206.782,Z 282.34,A -85,B 0,C 180,E1 -21259.869,E2 -21259.869} C_VEL
LIN {X 0,Y 206.76,Z 282.345,A -85,B 0,C 180,E1 -21264.072,E2 -21264.072} C_VEL
LIN {X 0,Y 206.733,Z 282.33,A -85,B 0,C 180,E1 -21268.42,E2 -21268.42} C_VEL
LIN {X 0,Y 206.711,Z 282.508,A -85,B 0,C 180,E1 -21272.871,E2 -21272.871} C_VEL
LIN {X 0,Y 208.946,Z 288.803,A -85,B 0,C 180,E1 -21277.26,E2 -21277.26} C_VEL
LIN {X 0,Y 210.936,Z 294.893,A -85,B 0,C 180,E1 -21280.941,E2 -21280.941} C_VEL
LIN {X 0,Y 211.346,Z 296.934,A -85,B 0,C 180,E1 -21281.842,E2 -21281.842} C_VEL
LIN {X 0,Y 211.618,Z 301.039,A -85,B 0,C 180,E1 -21282.996,E2 -21282.996} C_VEL
LIN {X 0,Y 212.16,Z 309.189,A -85,B 0,C 180,E1 -21284.558,E2 -21284.558} C_VEL
LIN {X 0,Y 213.258,Z 314.172,A -85,B 0,C 180,E1 -21285.413,E2 -21285.413} C_VEL
LIN {X 0,Y 215.536,Z 318.599,A -85,B 0,C 180,E1 -21286.282,E2 -21286.282} C_VEL
LIN {X 0,Y 222.056,Z 331.109,A -85,B 0,C 180,E1 -21288.273,E2 -21288.273} C_VEL
LIN {X 0,Y 228.367,Z 345.548,A -85,B 0,C 180,E1 -21290.149,E2 -21290.149} C_VEL
LIN {X 0,Y 229.09,Z 347.31,A -85,B 0,C 180,E1 -21290.358,E2 -21290.358} C_VEL
LIN {X 0,Y 224.676,Z 430.463,A -85,B 0,C 180,E1 -21292.907,E2 -21292.907} C_VEL
LIN {X 0,Y 223.144,Z 444.743,A -85,B 0,C 180,E1 -21293.666,E2 -21293.666} C_VEL
LIN {X 0,Y 221.309,Z 456.697,A -85,B 0,C 180,E1 -21294.582,E2 -21294.582} C_VEL
LIN {X 0,Y 218.63,Z 470.634,A -85,B 0,C 180,E1 -21296.047,E2 -21296.047} C_VEL
LIN {X 0,Y 215.746,Z 483.172,A -85,B 0,C 180,E1 -21297.794,E2 -21297.794} C_VEL
LIN {X 0,Y 212.493,Z 495.324,A -85,B 0,C 180,E1 -21299.984,E2 -21299.984} C_VEL
LIN {X 0,Y 209.035,Z 506.271,A -85,B 0,C 180,E1 -21302.466,E2 -21302.466} C_VEL
LIN {X 0,Y 205.928,Z 516.064,A -85,B 0,C 180,E1 -21305.288,E2 -21305.288} C_VEL
LIN {X 0,Y 203.309,Z 524.107,A -85,B 0,C 180,E1 -21308.186,E2 -21308.186} C_VEL
LIN {X 0,Y 201.078,Z 531.737,A -85,B 0,C 180,E1 -21311.666,E2 -21311.666} C_VEL
LIN {X 0,Y 199.428,Z 536.979,A -85,B 0,C 180,E1 -21314.675,E2 -21314.675} C_VEL
LIN {X 0,Y 198.253,Z 541.162,A -85,B 0,C 180,E1 -21317.72,E2 -21317.72} C_VEL
LIN {X 0,Y 197.47,Z 545.331,A -85,B 0,C 180,E1 -21321.816,E2 -21321.816} C_VEL
LIN {X 0,Y 197.267,Z 546.811,A -85,B 0,C 180,E1 -21323.865,E2 -21323.865} C_VEL
LIN {X 0,Y 197.235,Z 548.648,A -85,B 0,C 180,E1 -21327.958,E2 -21327.958} C_VEL
LIN {X 0,Y 197.362,Z 549.024,A -85,B 0,C 180,E1 -21330,E2 -21330} C_VEL
LIN {X 0,Y 197.244,Z 548.682,A -85,B 0,C 180,E1 -21334.087,E2 -21334.087} C_VEL
LIN {X 0,Y 197.482,Z 546.904,A -85,B 0,C 180,E1 -21338.184,E2 -21338.184} C_VEL
LIN {X 0,Y 198.346,Z 543.648,A -85,B 0,C 180,E1 -21342.275,E2 -21342.275} C_VEL
LIN {X 0,Y 199.542,Z 540.14,A -85,B 0,C 180,E1 -21345.317,E2 -21345.317} C_VEL
LIN {X 0,Y 201.207,Z 535.683,A -85,B 0,C 180,E1 -21348.322,E2 -21348.322} C_VEL
LIN {X 0,Y 203.651,Z 529.161,A -85,B 0,C 180,E1 -21351.775,E2 -21351.775} C_VEL
LIN {X 0,Y 206.362,Z 522.242,A -85,B 0,C 180,E1 -21354.657,E2 -21354.657} C_VEL
LIN {X 0,Y 209.556,Z 513.871,A -85,B 0,C 180,E1 -21357.46,E2 -21357.46} C_VEL
LIN {X 0,Y 213.338,Z 503.699,A -85,B 0,C 180,E1 -21360.157,E2 -21360.157} C_VEL
LIN {X 0,Y 216.993,Z 492.603,A -85,B 0,C 180,E1 -21362.473,E2 -21362.473} C_VEL
LIN {X 0,Y 220.049,Z 481.969,A -85,B 0,C 180,E1 -21364.257,E2 -21364.257} C_VEL
LIN {X 0,Y 223.221,Z 469.42,A -85,B 0,C 180,E1 -21365.901,E2 -21365.901} C_VEL
LIN {X 0,Y 225.989,Z 456.353,A -85,B 0,C 180,E1 -21367.191,E2 -21367.191} C_VEL
LIN {X 0,Y 228.236,Z 442.845,A -85,B 0,C 180,E1 -21368.153,E2 -21368.153} C_VEL
LIN {X 0,Y 229.749,Z 428.595,A -85,B 0,C 180,E1 -21368.835,E2 -21368.835} C_VEL
LIN {X 0,Y 233.996,Z 353.307,A -85,B 0,C 180,E1 -21371.072,E2 -21371.072} C_VEL
LIN {X 0,Y 233.751,Z 351.826,A -85,B 0,C 180,E1 -21371.185,E2 -21371.185} C_VEL
LIN {X 0,Y 227.794,Z 338.678,A -85,B 0,C 180,E1 -21373.063,E2 -21373.063} C_VEL
LIN {X 0,Y 220.759,Z 325.283,A -85,B 0,C 180,E1 -21375.385,E2 -21375.385} C_VEL
LIN {X 0,Y 215.182,Z 316.02,A -85,B 0,C 180,E1 -21377.342,E2 -21377.342} C_VEL
LIN {X 0,Y 209.437,Z 307.193,A -85,B 0,C 180,E1 -21379.513,E2 -21379.513} C_VEL
LIN {X 0,Y 206.595,Z 302.759,A -85,B 0,C 180,E1 -21380.765,E2 -21380.765} C_VEL
LIN {X 0,Y 204.828,Z 297.361,A -85,B 0,C 180,E1 -21384.318,E2 -21384.318} C_VEL
LIN {X 0,Y 202.791,Z 291.682,A -85,B 0,C 180,E1 -21388.679,E2 -21388.679} C_VEL
LIN {X 0,Y 201.081,Z 286.89,A -85,B 0,C 180,E1 -21392.977,E2 -21392.977} C_VEL
LIN {X 0,Y 199.748,Z 283.296,A -85,B 0,C 180,E1 -21397.026,E2 -21397.026} C_VEL
LIN {X 0,Y 199.794,Z 283.223,A -85,B 0,C 180,E1 -21401.758,E2 -21401.758} C_VEL
LIN {X 0,Y 199.833,Z 283.217,A -85,B 0,C 180,E1 -21405.749,E2 -21405.749} C_VEL
LIN {X 0,Y 200.068,Z 283.183,A -85,B 0,C 180,E1 -21409.885,E2 -21409.885} C_VEL
LIN {X 0,Y 200.031,Z 283.181,A -85,B 0,C 180,E1 -21413.95,E2 -21413.95} C_VEL
LIN {X 0,Y 200.319,Z 283.141,A -85,B 0,C 180,E1 -21417.99,E2 -21417.99} C_VEL
LIN {X 0,Y 200.477,Z 283.139,A -85,B 0,C 180,E1 -21420.001,E2 -21420.001} C_VEL
LIN {X 0,Y 200.029,Z 283.188,A -85,B 0,C 180,E1 -21424.03,E2 -21424.03} C_VEL
LIN {X 0,Y 200.11,Z 283.171,A -85,B 0,C 180,E1 -21428.077,E2 -21428.077} C_VEL
LIN {X 0,Y 199.884,Z 283.197,A -85,B 0,C 180,E1 -21432.18,E2 -21432.18} C_VEL
LIN {X 0,Y 199.802,Z 283.208,A -85,B 0,C 180,E1 -21436.344,E2 -21436.344} C_VEL
LIN {X 0,Y 199.741,Z 283.346,A -85,B 0,C 180,E1 -21441.141,E2 -21441.141} C_VEL
LIN {X 0,Y 201,Z 286.619,A -85,B 0,C 180,E1 -21444.809,E2 -21444.809} C_VEL
LIN {X 0,Y 203.155,Z 292.495,A -85,B 0,C 180,E1 -21450.135,E2 -21450.135} C_VEL
LIN {X 0,Y 205.176,Z 298.448,A -85,B 0,C 180,E1 -21454.707,E2 -21454.707} C_VEL
LIN {X 0,Y 207.233,Z 305.52,A -85,B 0,C 180,E1 -21459.339,E2 -21459.339} C_VEL
LIN {X 0,Y 208.063,Z 308.313,A -85,B 0,C 180,E1 -21460.865,E2 -21460.865} C_VEL
LIN {X 0,Y 211.209,Z 313.225,A -85,B 0,C 180,E1 -21462.122,E2 -21462.122} C_VEL
LIN {X 0,Y 215.454,Z 320.424,A -85,B 0,C 180,E1 -21463.713,E2 -21463.713} C_VEL
LIN {X 0,Y 220.097,Z 328.616,A -85,B 0,C 180,E1 -21465.348,E2 -21465.348} C_VEL
LIN {X 0,Y 226.753,Z 341.791,A -85,B 0,C 180,E1 -21467.55,E2 -21467.55} C_VEL
LIN {X 0,Y 230.677,Z 351.113,A -85,B 0,C 180,E1 -21468.81,E2 -21468.81} C_VEL
LIN {X 0,Y 232.937,Z 367.777,A -85,B 0,C 180,E1 -21469.936,E2 -21469.936} C_VEL
LIN {X 0,Y 229.776,Z 428.349,A -85,B 0,C 180,E1 -21471.658,E2 -21471.658} C_VEL
LIN {X 0,Y 228.193,Z 441.771,A -85,B 0,C 180,E1 -21472.327,E2 -21472.327} C_VEL
LIN {X 0,Y 226.182,Z 454.117,A -85,B 0,C 180,E1 -21473.264,E2 -21473.264} C_VEL
LIN {X 0,Y 223.666,Z 466.516,A -85,B 0,C 180,E1 -21474.569,E2 -21474.569} C_VEL
LIN {X 0,Y 221.054,Z 477.008,A -85,B 0,C 180,E1 -21476.008,E2 -21476.008} C_VEL
LIN {X 0,Y 217.826,Z 487.685,A -85,B 0,C 180,E1 -21477.835,E2 -21477.835} C_VEL
LIN {X 0,Y 214.253,Z 497.659,A -85,B 0,C 180,E1 -21479.985,E2 -21479.985} C_VEL
LIN {X 0,Y 210.528,Z 507.376,A -85,B 0,C 180,E1 -21482.677,E2 -21482.677} C_VEL
LIN {X 0,Y 207.186,Z 515.259,A -85,B 0,C 180,E1 -21485.447,E2 -21485.447} C_VEL
LIN {X 0,Y 204.439,Z 521.76,A -85,B 0,C 180,E1 -21488.371,E2 -21488.371} C_VEL
LIN {X 0,Y 201.909,Z 527.56,A -85,B 0,C 180,E1 -21491.744,E2 -21491.744} C_VEL
LIN {X 0,Y 200.061,Z 531.47,A -85,B 0,C 180,E1 -21494.724,E2 -21494.724} C_VEL
LIN {X 0,Y 198.868,Z 534.39,A -85,B 0,C 180,E1 -21497.758,E2 -21497.758} C_VEL
LIN {X 0,Y 198.238,Z 535.869,A -85,B 0,C 180,E1 -21499.79,E2 -21499.79} C_VEL
LIN {X 0,Y 197.509,Z 537.641,A -85,B 0,C 180,E1 -21503.872,E2 -21503.872} C_VEL
LIN {X 0,Y 197.339,Z 537.973,A -85,B 0,C 180,E1 -21507.959,E2 -21507.959} C_VEL
LIN {X 0,Y 197.542,Z 536.896,A -85,B 0,C 180,E1 -21512.039,E2 -21512.039} C_VEL
LIN {X 0,Y 197.806,Z 535.801,A -85,B 0,C 180,E1 -21514.075,E2 -21514.075} C_VEL
LIN {X 0,Y 198.727,Z 532.442,A -85,B 0,C 180,E1 -21518.132,E2 -21518.132} C_VEL
LIN {X 0,Y 199.885,Z 528.872,A -85,B 0,C 180,E1 -21521.15,E2 -21521.15} C_VEL
LIN {X 0,Y 201.466,Z 524.286,A -85,B 0,C 180,E1 -21524.134,E2 -21524.134} C_VEL
LIN {X 0,Y 203.973,Z 517.452,A -85,B 0,C 180,E1 -21527.546,E2 -21527.546} C_VEL
LIN {X 0,Y 206.585,Z 510.139,A -85,B 0,C 180,E1 -21530.408,E2 -21530.408} C_VEL
LIN {X 0,Y 209.645,Z 501.159,A -85,B 0,C 180,E1 -21533.197,E2 -21533.197} C_VEL
LIN {X 0,Y 212.875,Z 490.934,A -85,B 0,C 180,E1 -21535.678,E2 -21535.678} C_VEL
LIN {X 0,Y 215.737,Z 480.645,A -85,B 0,C 180,E1 -21537.659,E2 -21537.659} C_VEL
LIN {X 0,Y 218.595,Z 469.328,A -85,B 0,C 180,E1 -21539.359,E2 -21539.359} C_VEL
LIN {X 0,Y 221.117,Z 457.09,A -85,B 0,C 180,E1 -21540.78,E2 -21540.78} C_VEL
LIN {X 0,Y 222.934,Z 445.248,A -85,B 0,C 180,E1 -21541.82,E2 -21541.82} C_VEL
LIN {X 0,Y 224.464,Z 432.235,A -85,B 0,C 180,E1 -21542.595,E2 -21542.595} C_VEL
LIN {X 0,Y 225.435,Z 417.305,A -85,B 0,C 180,E1 -21543.124,E2 -21543.124} C_VEL
LIN {X 0,Y 227.813,Z 364.508,A -85,B 0,C 180,E1 -21544.639,E2 -21544.639} C_VEL
LIN {X 0,Y 224.829,Z 342.748,A -85,B 0,C 180,E1 -21546.037,E2 -21546.037} C_VEL
LIN {X 0,Y 218.19,Z 328.176,A -85,B 0,C 180,E1 -21548.03,E2 -21548.03} C_VEL
LIN {X 0,Y 212.191,Z 316.691,A -85,B 0,C 180,E1 -21549.921,E2 -21549.921} C_VEL
LIN {X 0,Y 207.534,Z 308.355,A -85,B 0,C 180,E1 -21551.561,E2 -21551.561} C_VEL
LIN {X 0,Y 205.474,Z 301.068,A -85,B 0,C 180,E1 -21555.479,E2 -21555.479} C_VEL
LIN {X 0,Y 203.106,Z 293.336,A -85,B 0,C 180,E1 -21560.289,E2 -21560.289} C_VEL
LIN {X 0,Y 201.16,Z 287.702,A -85,B 0,C 180,E1 -21564.28,E2 -21564.28} C_VEL
LIN {X 0,Y 199.691,Z 283.315,A -85,B 0,C 180,E1 -21567.828,E2 -21567.828} C_VEL
LIN {X 0,Y 199.686,Z 283.228,A -85,B 0,C 180,E1 -21572.771,E2 -21572.771} C_VEL
LIN {X 0,Y 199.737,Z 283.223,A -85,B 0,C 180,E1 -21577.228,E2 -21577.228} C_VEL
LIN {X 0,Y 199.795,Z 283.215,A -85,B 0,C 180,E1 -21581.757,E2 -21581.757} C_VEL
LIN {X 0,Y 199.832,Z 283.203,A -85,B 0,C 180,E1 -21585.747,E2 -21585.747} C_VEL
LIN {X 0,Y 200.02,Z 283.177,A -85,B 0,C 180,E1 -21589.881,E2 -21589.881} C_VEL
LIN {X 0,Y 200.023,Z 283.183,A -85,B 0,C 180,E1 -21593.949,E2 -21593.949} C_VEL
LIN {X 0,Y 200.317,Z 283.159,A -85,B 0,C 180,E1 -21597.989,E2 -21597.989} C_VEL
LIN {X 0,Y 200.476,Z 283.121,A -85,B 0,C 180,E1 -21599.999,E2 -21599.999} C_VEL
LIN {X 0,Y 200.028,Z 283.189,A -85,B 0,C 180,E1 -21604.029,E2 -21604.029} C_VEL
LIN {X 0,Y 200.108,Z 283.181,A -85,B 0,C 180,E1 -21608.075,E2 -21608.075} C_VEL
LIN {X 0,Y 200.033,Z 283.177,A -85,B 0,C 180,E1 -21610.347,E2 -21610.347} C_VEL
LIN {X 0,Y 199.8,Z 283.207,A -85,B 0,C 180,E1 -21616.343,E2 -21616.343} C_VEL
LIN {X 0,Y 199.699,Z 283.221,A -85,B 0,C 180,E1 -21620.605,E2 -21620.605} C_VEL
LIN {X 0,Y 199.669,Z 283.226,A -85,B 0,C 180,E1 -21624.984,E2 -21624.984} C_VEL
LIN {X 0,Y 199.661,Z 283.198,A -85,B 0,C 180,E1 -21629.524,E2 -21629.524} C_VEL
LIN {X 0,Y 199.684,Z 283.47,A -85,B 0,C 180,E1 -21630.393,E2 -21630.393} C_VEL
LIN {X 0,Y 201.887,Z 289.505,A -85,B 0,C 180,E1 -21635.056,E2 -21635.056} C_VEL
LIN {X 0,Y 204.182,Z 296.364,A -85,B 0,C 180,E1 -21639.551,E2 -21639.551} C_VEL
LIN {X 0,Y 206.201,Z 302.7,A -85,B 0,C 180,E1 -21643.123,E2 -21643.123} C_VEL
LIN {X 0,Y 212.422,Z 313.1,A -85,B 0,C 180,E1 -21645.29,E2 -21645.29} C_VEL
LIN {X 0,Y 215.536,Z 318.599,A -85,B 0,C 180,E1 -21646.282,E2 -21646.282} C_VEL
LIN {X 0,Y 217.262,Z 321.475,A -85,B 0,C 180,E1 -21646.806,E2 -21646.806} C_VEL
LIN {X 0,Y 219.015,Z 326.581,A -85,B 0,C 180,E1 -21647.418,E2 -21647.418} C_VEL
LIN {X 0,Y 220.059,Z 332.147,A -85,B 0,C 180,E1 -21647.888,E2 -21647.888} C_VEL
LIN {X 0,Y 221.742,Z 343.819,A -85,B 0,C 180,E1 -21648.744,E2 -21648.744} C_VEL
LIN {X 0,Y 222.677,Z 347.536,A -85,B 0,C 180,E1 -21649.095,E2 -21649.095} C_VEL
LIN {X 0,Y 223.355,Z 349.339,A -85,B 0,C 180,E1 -21649.309,E2 -21649.309} C_VEL
LIN {X 0,Y 218.923,Z 430.25,A -85,B 0,C 180,E1 -21651.835,E2 -21651.835} C_VEL
LIN {X 0,Y 217.343,Z 444.557,A -85,B 0,C 180,E1 -21652.606,E2 -21652.606} C_VEL
LIN {X 0,Y 215.33,Z 457.107,A -85,B 0,C 180,E1 -21653.587,E2 -21653.587} C_VEL
LIN {X 0,Y 212.736,Z 470.048,A -85,B 0,C 180,E1 -21654.971,E2 -21654.971} C_VEL
LIN {X 0,Y 209.976,Z 481.659,A -85,B 0,C 180,E1 -21656.593,E2 -21656.593} C_VEL
LIN {X 0,Y 206.626,Z 493.823,A -85,B 0,C 180,E1 -21658.756,E2 -21658.756} C_VEL
LIN {X 0,Y 203.369,Z 504.107,A -85,B 0,C 180,E1 -21661.066,E2 -21661.066} C_VEL
LIN {X 0,Y 199.957,Z 514.227,A -85,B 0,C 180,E1 -21663.939,E2 -21663.939} C_VEL
LIN {X 0,Y 197.098,Z 522.552,A -85,B 0,C 180,E1 -21666.907,E2 -21666.907} C_VEL
LIN {X 0,Y 194.737,Z 529.922,A -85,B 0,C 180,E1 -21670.215,E2 -21670.215} C_VEL
LIN {X 0,Y 192.529,Z 536.717,A -85,B 0,C 180,E1 -21674.111,E2 -21674.111} C_VEL
LIN {X 0,Y 191.253,Z 540.915,A -85,B 0,C 180,E1 -21677.263,E2 -21677.263} C_VEL
LIN {X 0,Y 190.426,Z 545.102,A -85,B 0,C 180,E1 -21681.511,E2 -21681.511} C_VEL
LIN {X 0,Y 190.194,Z 546.593,A -85,B 0,C 180,E1 -21683.636,E2 -21683.636} C_VEL
LIN {X 0,Y 190.141,Z 548.441,A -85,B 0,C 180,E1 -21687.882,E2 -21687.882} C_VEL
LIN {X 0,Y 190.264,Z 548.823,A -85,B 0,C 180,E1 -21690,E2 -21690} C_VEL
LIN {X 0,Y 190.16,Z 548.491,A -85,B 0,C 180,E1 -21694.239,E2 -21694.239} C_VEL
LIN {X 0,Y 190.441,Z 546.723,A -85,B 0,C 180,E1 -21698.489,E2 -21698.489} C_VEL
LIN {X 0,Y 191.349,Z 543.478,A -85,B 0,C 180,E1 -21702.731,E2 -21702.731} C_VEL
LIN {X 0,Y 193.223,Z 538.602,A -85,B 0,C 180,E1 -21706.916,E2 -21706.916} C_VEL
LIN {X 0,Y 195.128,Z 533.842,A -85,B 0,C 180,E1 -21710.009,E2 -21710.009} C_VEL
LIN {X 0,Y 197.897,Z 526.855,A -85,B 0,C 180,E1 -21713.548,E2 -21713.548} C_VEL
LIN {X 0,Y 201.522,Z 518.12,A -85,B 0,C 180,E1 -21716.96,E2 -21716.96} C_VEL
LIN {X 0,Y 205.162,Z 508.914,A -85,B 0,C 180,E1 -21719.782,E2 -21719.782} C_VEL
LIN {X 0,Y 208.983,Z 498.647,A -85,B 0,C 180,E1 -21722.267,E2 -21722.267} C_VEL
LIN {X 0,Y 212.619,Z 487.175,A -85,B 0,C 180,E1 -21724.475,E2 -21724.475} C_VEL
LIN {X 0,Y 216.237,Z 474.355,A -85,B 0,C 180,E1 -21726.38,E2 -21726.38} C_VEL
LIN {X 0,Y 219.474,Z 460.699,A -85,B 0,C 180,E1 -21727.909,E2 -21727.909} C_VEL
LIN {X 0,Y 221.942,Z 447.224,A -85,B 0,C 180,E1 -21729.002,E2 -21729.002} C_VEL
LIN {X 0,Y 223.821,Z 433.158,A -85,B 0,C 180,E1 -21729.774,E2 -21729.774} C_VEL
LIN {X 0,Y 225.24,Z 413.604,A -85,B 0,C 180,E1 -21730.422,E2 -21730.422} C_VEL
LIN {X 0,Y 228.555,Z 354.775,A -85,B 0,C 180,E1 -21732.193,E2 -21732.193} C_VEL
LIN {X 0,Y 223.312,Z 342.983,A -85,B 0,C 180,E1 -21733.938,E2 -21733.938} C_VEL
LIN {X 0,Y 216.5,Z 329.783,A -85,B 0,C 180,E1 -21736.305,E2 -21736.305} C_VEL
LIN {X 0,Y 211.421,Z 321.175,A -85,B 0,C 180,E1 -21738.18,E2 -21738.18} C_VEL
LIN {X 0,Y 205.781,Z 312.334,A -85,B 0,C 180,E1 -21740.42,E2 -21740.42} C_VEL
LIN {X 0,Y 202.116,Z 307.081,A -85,B 0,C 180,E1 -21741.976,E2 -21741.976} C_VEL
LIN {X 0,Y 199.487,Z 302.971,A -85,B 0,C 180,E1 -21743.286,E2 -21743.286} C_VEL
LIN {X 0,Y 197.477,Z 296.996,A -85,B 0,C 180,E1 -21747.736,E2 -21747.736} C_VEL
LIN {X 0,Y 195.617,Z 292.063,A -85,B 0,C 180,E1 -21752.157,E2 -21752.157} C_VEL
LIN {X 0,Y 194.145,Z 287.95,A -85,B 0,C 180,E1 -21756.535,E2 -21756.535} C_VEL
LIN {X 0,Y 192.769,Z 284.121,A -85,B 0,C 180,E1 -21761.983,E2 -21761.983} C_VEL
LIN {X 0,Y 192.807,Z 284.078,A -85,B 0,C 180,E1 -21767.368,E2 -21767.368} C_VEL
LIN {X 0,Y 193.059,Z 284.049,A -85,B 0,C 180,E1 -21771.628,E2 -21771.628} C_VEL
LIN {X 0,Y 193.261,Z 284.02,A -85,B 0,C 180,E1 -21777.917,E2 -21777.917} C_VEL
LIN {X 0,Y 193.441,Z 284.015,A -85,B 0,C 180,E1 -21780.001,E2 -21780.001} C_VEL
LIN {X 0,Y 192.976,Z 284.068,A -85,B 0,C 180,E1 -21784.178,E2 -21784.178} C_VEL
LIN {X 0,Y 193.06,Z 284.052,A -85,B 0,C 180,E1 -21788.374,E2 -21788.374} C_VEL
LIN {X 0,Y 192.807,Z 284.081,A -85,B 0,C 180,E1 -21792.634,E2 -21792.634} C_VEL
LIN {X 0,Y 192.778,Z 284.215,A -85,B 0,C 180,E1 -21796.413,E2 -21796.413} C_VEL
LIN {X 0,Y 194.056,Z 287.722,A -85,B 0,C 180,E1 -21801.234,E2 -21801.234} C_VEL
LIN {X 0,Y 195.251,Z 290.725,A -85,B 0,C 180,E1 -21804.637,E2 -21804.637} C_VEL
LIN {X 0,Y 197.246,Z 296.347,A -85,B 0,C 180,E1 -21809.924,E2 -21809.924} C_VEL
LIN {X 0,Y 199.106,Z 301.972,A -85,B 0,C 180,E1 -21814.387,E2 -21814.387} C_VEL
LIN {X 0,Y 200.907,Z 307.99,A -85,B 0,C 180,E1 -21818.384,E2 -21818.384} C_VEL
LIN {X 0,Y 203.977,Z 312.915,A -85,B 0,C 180,E1 -21819.778,E2 -21819.778} C_VEL
LIN {X 0,Y 208.432,Z 320.04,A -85,B 0,C 180,E1 -21821.609,E2 -21821.609} C_VEL
LIN {X 0,Y 213.785,Z 329.251,A -85,B 0,C 180,E1 -21823.66,E2 -21823.66} C_VEL
LIN {X 0,Y 220.257,Z 341.765,A -85,B 0,C 180,E1 -21825.967,E2 -21825.967} C_VEL
LIN {X 0,Y 225.5,Z 353.471,A -85,B 0,C 180,E1 -21827.733,E2 -21827.733} C_VEL
LIN {X 0,Y 227.525,Z 369.145,A -85,B 0,C 180,E1 -21828.823,E2 -21828.823} C_VEL
LIN {X 0,Y 224.288,Z 428.117,A -85,B 0,C 180,E1 -21830.517,E2 -21830.517} C_VEL
LIN {X 0,Y 222.635,Z 441.879,A -85,B 0,C 180,E1 -21831.215,E2 -21831.215} C_VEL
LIN {X 0,Y 220.326,Z 455.347,A -85,B 0,C 180,E1 -21832.263,E2 -21832.263} C_VEL
LIN {X 0,Y 217.674,Z 467.629,A -85,B 0,C 180,E1 -21833.611,E2 -21833.611} C_VEL
LIN {X 0,Y 214.573,Z 479.272,A -85,B 0,C 180,E1 -21835.302,E2 -21835.302} C_VEL
LIN {X 0,Y 210.67,Z 490.98,A -85,B 0,C 180,E1 -21837.458,E2 -21837.458} C_VEL
LIN {X 0,Y 206.783,Z 501.278,A -85,B 0,C 180,E1 -21839.914,E2 -21839.914} C_VEL
LIN {X 0,Y 203.042,Z 510.306,A -85,B 0,C 180,E1 -21842.702,E2 -21842.702} C_VEL
LIN {X 0,Y 199.698,Z 517.657,A -85,B 0,C 180,E1 -21845.574,E2 -21845.574} C_VEL
LIN {X 0,Y 196.603,Z 524.512,A -85,B 0,C 180,E1 -21849.055,E2 -21849.055} C_VEL
LIN {X 0,Y 194.473,Z 529.11,A -85,B 0,C 180,E1 -21852.111,E2 -21852.111} C_VEL
LIN {X 0,Y 192.693,Z 532.69,A -85,B 0,C 180,E1 -21855.208,E2 -21855.208} C_VEL
LIN {X 0,Y 191.24,Z 536.044,A -85,B 0,C 180,E1 -21859.412,E2 -21859.412} C_VEL
LIN {X 0,Y 190.431,Z 537.832,A -85,B 0,C 180,E1 -21863.643,E2 -21863.643} C_VEL
LIN {X 0,Y 190.246,Z 538.175,A -85,B 0,C 180,E1 -21867.883,E2 -21867.883} C_VEL
LIN {X 0,Y 190.451,Z 537.11,A -85,B 0,C 180,E1 -21872.115,E2 -21872.115} C_VEL
LIN {X 0,Y 190.729,Z 536.026,A -85,B 0,C 180,E1 -21874.226,E2 -21874.226} C_VEL
LIN {X 0,Y 191.715,Z 532.681,A -85,B 0,C 180,E1 -21878.432,E2 -21878.432} C_VEL
LIN {X 0,Y 192.928,Z 529.127,A -85,B 0,C 180,E1 -21881.557,E2 -21881.557} C_VEL
LIN {X 0,Y 194.611,Z 524.559,A -85,B 0,C 180,E1 -21884.642,E2 -21884.642} C_VEL
LIN {X 0,Y 197.216,Z 517.747,A -85,B 0,C 180,E1 -21888.168,E2 -21888.168} C_VEL
LIN {X 0,Y 199.966,Z 510.458,A -85,B 0,C 180,E1 -21891.115,E2 -21891.115} C_VEL
LIN {X 0,Y 203.16,Z 501.508,A -85,B 0,C 180,E1 -21893.983,E2 -21893.983} C_VEL
LIN {X 0,Y 206.522,Z 491.348,A -85,B 0,C 180,E1 -21896.528,E2 -21896.528} C_VEL
LIN {X 0,Y 209.496,Z 481.119,A -85,B 0,C 180,E1 -21898.557,E2 -21898.557} C_VEL
LIN {X 0,Y 212.443,Z 469.978,A -85,B 0,C 180,E1 -21900.28,E2 -21900.28} C_VEL
LIN {X 0,Y 215.079,Z 457.763,A -85,B 0,C 180,E1 -21901.743,E2 -21901.743} C_VEL
LIN {X 0,Y 217.046,Z 445.594,A -85,B 0,C 180,E1 -21902.844,E2 -21902.844} C_VEL
LIN {X 0,Y 218.648,Z 432.59,A -85,B 0,C 180,E1 -21903.643,E2 -21903.643} C_VEL
LIN {X 0,Y 219.663,Z 417.761,A -85,B 0,C 180,E1 -21904.183,E2 -21904.183} C_VEL
LIN {X 0,Y 222.107,Z 365.145,A -85,B 0,C 180,E1 -21905.731,E2 -21905.731} C_VEL
LIN {X 0,Y 219.535,Z 345.675,A -85,B 0,C 180,E1 -21907.024,E2 -21907.024} C_VEL
LIN {X 0,Y 212.685,Z 330.519,A -85,B 0,C 180,E1 -21909.204,E2 -21909.204} C_VEL
LIN {X 0,Y 207.131,Z 319.937,A -85,B 0,C 180,E1 -21911.061,E2 -21911.061} C_VEL
LIN {X 0,Y 202.25,Z 311.666,A -85,B 0,C 180,E1 -21912.78,E2 -21912.78} C_VEL
LIN {X 0,Y 200.284,Z 308.034,A -85,B 0,C 180,E1 -21913.636,E2 -21913.636} C_VEL
LIN {X 0,Y 198.285,Z 301.181,A -85,B 0,C 180,E1 -21917.666,E2 -21917.666} C_VEL
LIN {X 0,Y 196.341,Z 294.818,A -85,B 0,C 180,E1 -21921.95,E2 -21921.95} C_VEL
LIN {X 0,Y 194.404,Z 289.226,A -85,B 0,C 180,E1 -21926.25,E2 -21926.25} C_VEL
LIN {X 0,Y 192.656,Z 284.165,A -85,B 0,C 180,E1 -21930.857,E2 -21930.857} C_VEL
LIN {X 0,Y 192.704,Z 284.093,A -85,B 0,C 180,E1 -21936.348,E2 -21936.348} C_VEL
LIN {X 0,Y 192.73,Z 284.092,A -85,B 0,C 180,E1 -21941.457,E2 -21941.457} C_VEL
LIN {X 0,Y 192.76,Z 284.082,A -85,B 0,C 180,E1 -21945.213,E2 -21945.213} C_VEL
LIN {X 0,Y 192.943,Z 284.059,A -85,B 0,C 180,E1 -21949.566,E2 -21949.566} C_VEL
LIN {X 0,Y 193.038,Z 284.054,A -85,B 0,C 180,E1 -21951.626,E2 -21951.626} C_VEL
LIN {X 0,Y 193.259,Z 284.038,A -85,B 0,C 180,E1 -21957.915,E2 -21957.915} C_VEL
LIN {X 0,Y 193.44,Z 283.997,A -85,B 0,C 180,E1 -21959.999,E2 -21959.999} C_VEL
LIN {X 0,Y 192.974,Z 284.065,A -85,B 0,C 180,E1 -21964.176,E2 -21964.176} C_VEL
LIN {X 0,Y 193.059,Z 284.061,A -85,B 0,C 180,E1 -21968.372,E2 -21968.372} C_VEL
LIN {X 0,Y 192.806,Z 284.084,A -85,B 0,C 180,E1 -21972.632,E2 -21972.632} C_VEL
LIN {X 0,Y 192.753,Z 284.087,A -85,B 0,C 180,E1 -21976.958,E2 -21976.958} C_VEL
LIN {X 0,Y 192.635,Z 284.103,A -85,B 0,C 180,E1 -21981.397,E2 -21981.397} C_VEL
LIN {X 0,Y 192.661,Z 284.1,A -85,B 0,C 180,E1 -21984.224,E2 -21984.224} C_VEL
LIN {X 0,Y 192.69,Z 284.308,A -85,B 0,C 180,E1 -21987.417,E2 -21987.417} C_VEL
LIN {X 0,Y 194.89,Z 290.465,A -85,B 0,C 180,E1 -21992.746,E2 -21992.746} C_VEL
LIN {X 0,Y 196.518,Z 295.093,A -85,B 0,C 180,E1 -21996.162,E2 -21996.162} C_VEL
LIN {X 0,Y 198.958,Z 302.687,A -85,B 0,C 180,E1 -22000.987,E2 -22000.987} C_VEL
LIN {X 0,Y 202.739,Z 308.863,A -85,B 0,C 180,E1 -22002.529,E2 -22002.529} C_VEL
LIN {X 0,Y 208.561,Z 318.527,A -85,B 0,C 180,E1 -22004.566,E2 -22004.566} C_VEL
LIN {X 0,Y 215.213,Z 330.904,A -85,B 0,C 180,E1 -22006.746,E2 -22006.746} C_VEL
LIN {X 0,Y 221.806,Z 345.396,A -85,B 0,C 180,E1 -22008.824,E2 -22008.824} C_VEL
LIN {X 0,Y 222.677,Z 347.536,A -85,B 0,C 180,E1 -22009.095,E2 -22009.095} C_VEL
LIN {X 0,Y 223.198,Z 351.176,A -85,B 0,C 180,E1 -22009.354,E2 -22009.354} C_VEL
LIN {X 0,Y 222.693,Z 355.975,A -85,B 0,C 180,E1 -22009.451,E2 -22009.451} C_VEL
LIN {X 0,Y 220.729,Z 362.629,A -85,B 0,C 180,E1 -22009.328,E2 -22009.328} C_VEL
LIN {X 0,Y 217.286,Z 372.439,A -85,B 0,C 180,E1 -22009.027,E2 -22009.027} C_VEL
LIN {X 0,Y 216.322,Z 377.505,A -85,B 0,C 180,E1 -22009.04,E2 -22009.04} C_VEL
LIN {X 0,Y 216.252,Z 378.529,A -85,B 0,C 180,E1 -22009.07,E2 -22009.07} C_VEL
LIN {X 0,Y 213.194,Z 430.613,A -85,B 0,C 180,E1 -22010.733,E2 -22010.733} C_VEL
LIN {X 0,Y 211.62,Z 444.372,A -85,B 0,C 180,E1 -22011.488,E2 -22011.488} C_VEL
LIN {X 0,Y 209.424,Z 457.517,A -85,B 0,C 180,E1 -22012.538,E2 -22012.538} C_VEL
LIN {X 0,Y 206.95,Z 469.465,A -85,B 0,C 180,E1 -22013.84,E2 -22013.84} C_VEL
LIN {X 0,Y 203.814,Z 482.032,A -85,B 0,C 180,E1 -22015.624,E2 -22015.624} C_VEL
LIN {X 0,Y 200.491,Z 493.62,A -85,B 0,C 180,E1 -22017.742,E2 -22017.742} C_VEL
LIN {X 0,Y 197.138,Z 503.744,A -85,B 0,C 180,E1 -22020.06,E2 -22020.06} C_VEL
LIN {X 0,Y 193.561,Z 513.899,A -85,B 0,C 180,E1 -22023.009,E2 -22023.009} C_VEL
LIN {X 0,Y 190.518,Z 522.25,A -85,B 0,C 180,E1 -22026.061,E2 -22026.061} C_VEL
LIN {X 0,Y 188.053,Z 529.39,A -85,B 0,C 180,E1 -22029.341,E2 -22029.341} C_VEL
LIN {X 0,Y 186.206,Z 534.807,A -85,B 0,C 180,E1 -22032.426,E2 -22032.426} C_VEL
LIN {X 0,Y 184.678,Z 539.397,A -85,B 0,C 180,E1 -22035.679,E2 -22035.679} C_VEL
LIN {X 0,Y 183.759,Z 542.97,A -85,B 0,C 180,E1 -22038.976,E2 -22038.976} C_VEL
LIN {X 0,Y 183.372,Z 544.871,A -85,B 0,C 180,E1 -22041.182,E2 -22041.182} C_VEL
LIN {X 0,Y 183.012,Z 547.485,A -85,B 0,C 180,E1 -22045.595,E2 -22045.595} C_VEL
LIN {X 0,Y 183.168,Z 548.621,A -85,B 0,C 180,E1 -22050,E2 -22050} C_VEL
LIN {X 0,Y 183.073,Z 548.299,A -85,B 0,C 180,E1 -22054.403,E2 -22054.403} C_VEL
LIN {X 0,Y 183.389,Z 546.541,A -85,B 0,C 180,E1 -22058.818,E2 -22058.818} C_VEL
LIN {X 0,Y 184.37,Z 543.307,A -85,B 0,C 180,E1 -22063.221,E2 -22063.221} C_VEL
LIN {X 0,Y 186.386,Z 538.443,A -85,B 0,C 180,E1 -22067.557,E2 -22067.557} C_VEL
LIN {X 0,Y 188.901,Z 532.319,A -85,B 0,C 180,E1 -22071.548,E2 -22071.548} C_VEL
LIN {X 0,Y 191.845,Z 525.58,A -85,B 0,C 180,E1 -22074.916,E2 -22074.916} C_VEL
LIN {X 0,Y 195.177,Z 517.986,A -85,B 0,C 180,E1 -22077.911,E2 -22077.911} C_VEL
LIN {X 0,Y 199.022,Z 508.786,A -85,B 0,C 180,E1 -22080.799,E2 -22080.799} C_VEL
LIN {X 0,Y 203.004,Z 498.524,A -85,B 0,C 180,E1 -22083.339,E2 -22083.339} C_VEL
LIN {X 0,Y 206.805,Z 487.056,A -85,B 0,C 180,E1 -22085.589,E2 -22085.589} C_VEL
LIN {X 0,Y 210.56,Z 474.234,A -85,B 0,C 180,E1 -22087.527,E2 -22087.527} C_VEL
LIN {X 0,Y 213.907,Z 460.57,A -85,B 0,C 180,E1 -22089.08,E2 -22089.08} C_VEL
LIN {X 0,Y 216.483,Z 447.071,A -85,B 0,C 180,E1 -22090.182,E2 -22090.182} C_VEL
LIN {X 0,Y 218.423,Z 432.95,A -85,B 0,C 180,E1 -22090.963,E2 -22090.963} C_VEL
LIN {X 0,Y 219.895,Z 413.291,A -85,B 0,C 180,E1 -22091.619,E2 -22091.619} C_VEL
LIN {X 0,Y 223.188,Z 357.008,A -85,B 0,C 180,E1 -22093.337,E2 -22093.337} C_VEL
LIN {X 0,Y 217.908,Z 345.22,A -85,B 0,C 180,E1 -22095.197,E2 -22095.197} C_VEL
LIN {X 0,Y 211.929,Z 333.646,A -85,B 0,C 180,E1 -22097.4,E2 -22097.4} C_VEL
LIN {X 0,Y 205.866,Z 323.179,A -85,B 0,C 180,E1 -22099.802,E2 -22099.802} C_VEL
LIN {X 0,Y 199.217,Z 313.05,A -85,B 0,C 180,E1 -22102.682,E2 -22102.682} C_VEL
LIN {X 0,Y 195.309,Z 307.578,A -85,B 0,C 180,E1 -22104.533,E2 -22104.533} C_VEL
LIN {X 0,Y 192.401,Z 303.217,A -85,B 0,C 180,E1 -22106.149,E2 -22106.149} C_VEL
LIN {X 0,Y 190.741,Z 298.4,A -85,B 0,C 180,E1 -22110.171,E2 -22110.171} C_VEL
LIN {X 0,Y 189.486,Z 294.935,A -85,B 0,C 180,E1 -22113.572,E2 -22113.572} C_VEL
LIN {X 0,Y 187.934,Z 291.209,A -85,B 0,C 180,E1 -22118.041,E2 -22118.041} C_VEL
LIN {X 0,Y 186.896,Z 288.12,A -85,B 0,C 180,E1 -22122.493,E2 -22122.493} C_VEL
LIN {X 0,Y 185.922,Z 284.987,A -85,B 0,C 180,E1 -22129.36,E2 -22129.36} C_VEL
LIN {X 0,Y 185.958,Z 284.93,A -85,B 0,C 180,E1 -22133.49,E2 -22133.49} C_VEL
LIN {X 0,Y 186.205,Z 284.898,A -85,B 0,C 180,E1 -22137.838,E2 -22137.838} C_VEL
LIN {X 0,Y 186.404,Z 284.891,A -85,B 0,C 180,E1 -22140.001,E2 -22140.001} C_VEL
LIN {X 0,Y 185.924,Z 284.948,A -85,B 0,C 180,E1 -22144.336,E2 -22144.336} C_VEL
LIN {X 0,Y 185.978,Z 285.024,A -85,B 0,C 180,E1 -22149.246,E2 -22149.246} C_VEL
LIN {X 0,Y 186.818,Z 287.964,A -85,B 0,C 180,E1 -22155.269,E2 -22155.269} C_VEL
LIN {X 0,Y 188.389,Z 292.013,A -85,B 0,C 180,E1 -22161.152,E2 -22161.152} C_VEL
LIN {X 0,Y 189.653,Z 295.623,A -85,B 0,C 180,E1 -22165.225,E2 -22165.225} C_VEL
LIN {X 0,Y 191.345,Z 300.234,A -85,B 0,C 180,E1 -22169.727,E2 -22169.727} C_VEL
LIN {X 0,Y 193.384,Z 306.678,A -85,B 0,C 180,E1 -22174.918,E2 -22174.918} C_VEL
LIN {X 0,Y 193.891,Z 308.069,A -85,B 0,C 180,E1 -22175.672,E2 -22175.672} C_VEL
LIN {X 0,Y 197.157,Z 312.926,A -85,B 0,C 180,E1 -22177.301,E2 -22177.301} C_VEL
LIN {X 0,Y 202.244,Z 321.105,A -85,B 0,C 180,E1 -22179.626,E2 -22179.626} C_VEL
LIN {X 0,Y 205.64,Z 326.653,A -85,B 0,C 180,E1 -22181.06,E2 -22181.06} C_VEL
LIN {X 0,Y 211.59,Z 337.354,A -85,B 0,C 180,E1 -22183.419,E2 -22183.419} C_VEL
LIN {X 0,Y 217.835,Z 350.232,A -85,B 0,C 180,E1 -22185.713,E2 -22185.713} C_VEL
LIN {X 0,Y 220.563,Z 356.917,A -85,B 0,C 180,E1 -22186.69,E2 -22186.69} C_VEL
LIN {X 0,Y 222.196,Z 370.507,A -85,B 0,C 180,E1 -22187.654,E2 -22187.654} C_VEL
LIN {X 0,Y 218.885,Z 427.969,A -85,B 0,C 180,E1 -22189.323,E2 -22189.323} C_VEL
LIN {X 0,Y 217.282,Z 441.217,A -85,B 0,C 180,E1 -22189.996,E2 -22189.996} C_VEL
LIN {X 0,Y 214.983,Z 454.311,A -85,B 0,C 180,E1 -22191.002,E2 -22191.002} C_VEL
LIN {X 0,Y 212.42,Z 465.999,A -85,B 0,C 180,E1 -22192.261,E2 -22192.261} C_VEL
LIN {X 0,Y 209.593,Z 476.616,A -85,B 0,C 180,E1 -22193.745,E2 -22193.745} C_VEL
LIN {X 0,Y 205.941,Z 487.892,A -85,B 0,C 180,E1 -22195.731,E2 -22195.731} C_VEL
LIN {X 0,Y 202.085,Z 497.882,A -85,B 0,C 180,E1 -22197.971,E2 -22197.971} C_VEL
LIN {X 0,Y 198.625,Z 506.145,A -85,B 0,C 180,E1 -22200.307,E2 -22200.307} C_VEL
LIN {X 0,Y 194.893,Z 514.3,A -85,B 0,C 180,E1 -22203.208,E2 -22203.208} C_VEL
LIN {X 0,Y 191.362,Z 521.779,A -85,B 0,C 180,E1 -22206.66,E2 -22206.66} C_VEL
LIN {X 0,Y 188.438,Z 527.865,A -85,B 0,C 180,E1 -22210.387,E2 -22210.387} C_VEL
LIN {X 0,Y 185.797,Z 532.854,A -85,B 0,C 180,E1 -22214.646,E2 -22214.646} C_VEL
LIN {X 0,Y 184.233,Z 536.219,A -85,B 0,C 180,E1 -22219.004,E2 -22219.004} C_VEL
LIN {X 0,Y 183.377,Z 538.022,A -85,B 0,C 180,E1 -22223.398,E2 -22223.398} C_VEL
LIN {X 0,Y 183.154,Z 538.377,A -85,B 0,C 180,E1 -22227.801,E2 -22227.801} C_VEL
LIN {X 0,Y 183.362,Z 537.323,A -85,B 0,C 180,E1 -22232.196,E2 -22232.196} C_VEL
LIN {X 0,Y 183.656,Z 536.25,A -85,B 0,C 180,E1 -22234.389,E2 -22234.389} C_VEL
LIN {X 0,Y 184.695,Z 532.921,A -85,B 0,C 180,E1 -22238.755,E2 -22238.755} C_VEL
LIN {X 0,Y 185.999,Z 529.382,A -85,B 0,C 180,E1 -22241.994,E2 -22241.994} C_VEL
LIN {X 0,Y 187.751,Z 524.832,A -85,B 0,C 180,E1 -22245.19,E2 -22245.19} C_VEL
LIN {X 0,Y 190.485,Z 518.042,A -85,B 0,C 180,E1 -22248.834,E2 -22248.834} C_VEL
LIN {X 0,Y 193.386,Z 510.777,A -85,B 0,C 180,E1 -22251.87,E2 -22251.87} C_VEL
LIN {X 0,Y 196.696,Z 501.859,A -85,B 0,C 180,E1 -22254.823,E2 -22254.823} C_VEL
LIN {X 0,Y 200.221,Z 491.762,A -85,B 0,C 180,E1 -22257.432,E2 -22257.432} C_VEL
LIN {X 0,Y 203.311,Z 481.592,A -85,B 0,C 180,E1 -22259.51,E2 -22259.51} C_VEL
LIN {X 0,Y 206.348,Z 470.624,A -85,B 0,C 180,E1 -22261.257,E2 -22261.257} C_VEL
LIN {X 0,Y 209.108,Z 458.436,A -85,B 0,C 180,E1 -22262.761,E2 -22262.761} C_VEL
LIN {X 0,Y 211.336,Z 445.145,A -85,B 0,C 180,E1 -22263.992,E2 -22263.992} C_VEL
LIN {X 0,Y 213.021,Z 431.867,A -85,B 0,C 180,E1 -22264.793,E2 -22264.793} C_VEL
LIN {X 0,Y 214.185,Z 414.8,A -85,B 0,C 180,E1 -22265.391,E2 -22265.391} C_VEL
LIN {X 0,Y 216.524,Z 366.393,A -85,B 0,C 180,E1 -22266.847,E2 -22266.847} C_VEL
LIN {X 0,Y 214.269,Z 348.48,A -85,B 0,C 180,E1 -22268.074,E2 -22268.074} C_VEL
LIN {X 0,Y 207.522,Z 333.57,A -85,B 0,C 180,E1 -22270.346,E2 -22270.346} C_VEL
LIN {X 0,Y 201.602,Z 322.211,A -85,B 0,C 180,E1 -22272.46,E2 -22272.46} C_VEL
LIN {X 0,Y 195.868,Z 312.568,A -85,B 0,C 180,E1 -22274.644,E2 -22274.644} C_VEL
LIN {X 0,Y 193.117,Z 307.856,A -85,B 0,C 180,E1 -22275.891,E2 -22275.891} C_VEL
LIN {X 0,Y 190.937,Z 300.565,A -85,B 0,C 180,E1 -22280.619,E2 -22280.619} C_VEL
LIN {X 0,Y 189.179,Z 295.02,A -85,B 0,C 180,E1 -22284.814,E2 -22284.814} C_VEL
LIN {X 0,Y 187.736,Z 290.832,A -85,B 0,C 180,E1 -22288.391,E2 -22288.391} C_VEL
LIN {X 0,Y 186.329,Z 287.309,A -85,B 0,C 180,E1 -22291.869,E2 -22291.869} C_VEL
LIN {X 0,Y 185.561,Z 285.055,A -85,B 0,C 180,E1 -22294.51,E2 -22294.51} C_VEL
LIN {X 0,Y 185.596,Z 284.99,A -85,B 0,C 180,E1 -22297.748,E2 -22297.748} C_VEL
LIN {X 0,Y 185.688,Z 284.979,A -85,B 0,C 180,E1 -22302.374,E2 -22302.374} C_VEL
LIN {X 0,Y 185.726,Z 284.969,A -85,B 0,C 180,E1 -22306.876,E2 -22306.876} C_VEL
LIN {X 0,Y 185.984,Z 284.929,A -85,B 0,C 180,E1 -22311.305,E2 -22311.305} C_VEL
LIN {X 0,Y 186.203,Z 284.916,A -85,B 0,C 180,E1 -22317.836,E2 -22317.836} C_VEL
LIN {X 0,Y 186.403,Z 284.873,A -85,B 0,C 180,E1 -22319.999,E2 -22319.999} C_VEL
LIN {X 0,Y 185.921,Z 284.941,A -85,B 0,C 180,E1 -22324.335,E2 -22324.335} C_VEL
LIN {X 0,Y 186.006,Z 284.94,A -85,B 0,C 180,E1 -22328.692,E2 -22328.692} C_VEL
LIN {X 0,Y 185.73,Z 284.971,A -85,B 0,C 180,E1 -22333.122,E2 -22333.122} C_VEL
LIN {X 0,Y 185.687,Z 284.974,A -85,B 0,C 180,E1 -22337.625,E2 -22337.625} C_VEL
LIN {X 0,Y 185.67,Z 285.167,A -85,B 0,C 180,E1 -22343.862,E2 -22343.862} C_VEL
LIN {X 0,Y 187.051,Z 289.175,A -85,B 0,C 180,E1 -22348.011,E2 -22348.011} C_VEL
LIN {X 0,Y 188.995,Z 294.425,A -85,B 0,C 180,E1 -22352.628,E2 -22352.628} C_VEL
LIN {X 0,Y 190.589,Z 299.076,A -85,B 0,C 180,E1 -22356.156,E2 -22356.156} C_VEL
LIN {X 0,Y 191.973,Z 303.228,A -85,B 0,C 180,E1 -22358.813,E2 -22358.813} C_VEL
LIN {X 0,Y 196.873,Z 310.879,A -85,B 0,C 180,E1 -22360.891,E2 -22360.891} C_VEL
LIN {X 0,Y 202.506,Z 320.015,A -85,B 0,C 180,E1 -22363.013,E2 -22363.013} C_VEL
LIN {X 0,Y 209.474,Z 332.85,A -85,B 0,C 180,E1 -22365.458,E2 -22365.458} C_VEL
LIN {X 0,Y 215.188,Z 345.268,A -85,B 0,C 180,E1 -22367.38,E2 -22367.38} C_VEL
LIN {X 0,Y 217.773,Z 351.417,A -85,B 0,C 180,E1 -22368.223,E2 -22368.223} C_VEL
LIN {X 0,Y 216.252,Z 378.529,A -85,B 0,C 180,E1 -22369.07,E2 -22369.07} C_VEL
LIN {X 0,Y 215.457,Z 384.368,A -85,B 0,C 180,E1 -22369.152,E2 -22369.152} C_VEL
LIN {X 0,Y 209.86,Z 403.358,A -85,B 0,C 180,E1 -22368.768,E2 -22368.768} C_VEL
LIN {X 0,Y 208.951,Z 409.204,A -85,B 0,C 180,E1 -22368.827,E2 -22368.827} C_VEL
LIN {X 0,Y 207.44,Z 431.742,A -85,B 0,C 180,E1 -22369.599,E2 -22369.599} C_VEL
LIN {X 0,Y 205.738,Z 445.707,A -85,B 0,C 180,E1 -22370.41,E2 -22370.41} C_VEL
LIN {X 0,Y 203.596,Z 457.929,A -85,B 0,C 180,E1 -22371.428,E2 -22371.428} C_VEL
LIN {X 0,Y 200.812,Z 470.655,A -85,B 0,C 180,E1 -22372.865,E2 -22372.865} C_VEL
LIN {X 0,Y 197.574,Z 482.965,A -85,B 0,C 180,E1 -22374.688,E2 -22374.688} C_VEL
LIN {X 0,Y 194.422,Z 493.417,A -85,B 0,C 180,E1 -22376.665,E2 -22376.665} C_VEL
LIN {X 0,Y 190.993,Z 503.376,A -85,B 0,C 180,E1 -22378.993,E2 -22378.993} C_VEL
LIN {X 0,Y 187.756,Z 512.028,A -85,B 0,C 180,E1 -22381.495,E2 -22381.495} C_VEL
LIN {X 0,Y 184.488,Z 520.694,A -85,B 0,C 180,E1 -22384.624,E2 -22384.624} C_VEL
LIN {X 0,Y 181.406,Z 528.859,A -85,B 0,C 180,E1 -22388.403,E2 -22388.403} C_VEL
LIN {X 0,Y 179.388,Z 534.546,A -85,B 0,C 180,E1 -22391.735,E2 -22391.735} C_VEL
LIN {X 0,Y 177.754,Z 539.149,A -85,B 0,C 180,E1 -22395.109,E2 -22395.109} C_VEL
LIN {X 0,Y 176.731,Z 542.731,A -85,B 0,C 180,E1 -22398.532,E2 -22398.532} C_VEL
LIN {X 0,Y 176.317,Z 544.639,A -85,B 0,C 180,E1 -22400.826,E2 -22400.826} C_VEL
LIN {X 0,Y 176.044,Z 546.152,A -85,B 0,C 180,E1 -22403.122,E2 -22403.122} C_VEL
LIN {X 0,Y 175.948,Z 548.027,A -85,B 0,C 180,E1 -22407.711,E2 -22407.711} C_VEL
LIN {X 0,Y 176.075,Z 548.42,A -85,B 0,C 180,E1 -22410,E2 -22410} C_VEL
LIN {X 0,Y 175.969,Z 548.108,A -85,B 0,C 180,E1 -22414.582,E2 -22414.582} C_VEL
LIN {X 0,Y 176.334,Z 546.359,A -85,B 0,C 180,E1 -22419.173,E2 -22419.173} C_VEL
LIN {X 0,Y 177.411,Z 543.137,A -85,B 0,C 180,E1 -22423.75,E2 -22423.75} C_VEL
LIN {X 0,Y 178.955,Z 539.65,A -85,B 0,C 180,E1 -22427.13,E2 -22427.13} C_VEL
LIN {X 0,Y 180.976,Z 535.219,A -85,B 0,C 180,E1 -22430.457,E2 -22430.457} C_VEL
LIN {X 0,Y 183.867,Z 528.721,A -85,B 0,C 180,E1 -22434.261,E2 -22434.261} C_VEL
LIN {X 0,Y 187.661,Z 520.576,A -85,B 0,C 180,E1 -22437.913,E2 -22437.913} C_VEL
LIN {X 0,Y 191.481,Z 511.941,A -85,B 0,C 180,E1 -22440.92,E2 -22440.92} C_VEL
LIN {X 0,Y 195.949,Z 501.368,A -85,B 0,C 180,E1 -22443.774,E2 -22443.774} C_VEL
LIN {X 0,Y 200.056,Z 489.87,A -85,B 0,C 180,E1 -22446.24,E2 -22446.24} C_VEL
LIN {X 0,Y 203.643,Z 478.749,A -85,B 0,C 180,E1 -22448.089,E2 -22448.089} C_VEL
LIN {X 0,Y 206.815,Z 467.284,A -85,B 0,C 180,E1 -22449.58,E2 -22449.58} C_VEL
LIN {X 0,Y 209.653,Z 454.828,A -85,B 0,C 180,E1 -22450.819,E2 -22450.819} C_VEL
LIN {X 0,Y 212.004,Z 441.584,A -85,B 0,C 180,E1 -22451.761,E2 -22451.761} C_VEL
LIN {X 0,Y 213.648,Z 426.982,A -85,B 0,C 180,E1 -22452.449,E2 -22452.449} C_VEL
LIN {X 0,Y 217.889,Z 359.305,A -85,B 0,C 180,E1 -22454.541,E2 -22454.541} C_VEL
LIN {X 0,Y 212.854,Z 348.057,A -85,B 0,C 180,E1 -22456.424,E2 -22456.424} C_VEL
LIN {X 0,Y 206.79,Z 336.168,A -85,B 0,C 180,E1 -22458.815,E2 -22458.815} C_VEL
LIN {X 0,Y 199.605,Z 324.068,A -85,B 0,C 180,E1 -22461.892,E2 -22461.892} C_VEL
LIN {X 0,Y 195.217,Z 317.574,A -85,B 0,C 180,E1 -22463.942,E2 -22463.942} C_VEL
LIN {X 0,Y 192.185,Z 313.156,A -85,B 0,C 180,E1 -22465.472,E2 -22465.472} C_VEL
